# B&R Automation Studio project TD52 (part 134)

#### MsgSYCyclic.st
```iecst
(*******************************************************************************
MsgSY	 			 messages

This code is confidential and proprietary to the INNIO Company.
It may not be used in any form, or reproduced in any manner,
without written permission of the INNIO Company.
Copyright, INNIO Company, 2022

Customized modifications: -
------------------------

History:
-------
V2.12	24.04.2006	LH			adapted for esy new
V2.20	07.02.2007	LH			adapted for supporting customer mcb
		26.04.2007	LH			closing failure gcb (5th try was successful):
					               - gcb on + 10 sec --> reset counter
					               - dalay closing fail. = 11 sec
		09.05.2007	LH			0/1-sign. fail. mcbx: activation with RUN in case of old hardware
V2.30	18.01.2008	LH			adapted for test-bench run
		14.02.2008	LH			reset moved from end to begin
		28.03.2008	LH			gcb not closed and load > 10% --> gcb position failure
		07.04.2008	LH			new gcb position monitoring active with release from engine control
V2.311a	13.05.2008	LH			set delay time new gcb position failure up to 2 sec.
V2.33.0	16.07.2008	lettenb.	mcb[1].alm_psf disabled with PRF_I (circuitus)
V2.60.0	13.08.2009	lettenb.	ton_gcb_opf	for opening mcb with delay addedf
V3.20.0	14.04.2010	lettenb.	change to new global structure ALM
		11.11.2010				1216 enable busbar 1 voltage sensor failure	if not bSynch
		07.12.2010				1219 ctd_gcb_cf[1].LOAD	mit quitt_wa
								(reset ctd_gcb_cf[1] funktioniert nicht wenn eng[1].sy_rdy = false)
V3.99.0	25.02.2012	lettenb.	3329,3352,3575,3576,3577 added (integration V3.30-V3.40)
		24.05.2013				reset OUT_xx.txx2AB.bGnlTripx changed
		18.06.2013				2140 removed (made in MM_OP), 2139 logic changed, xMsg2139+xMsg2140 removed
V4.00.0	27.02.2014				logger added
		06.03.2014				Para.bGlowIgnPrevent -> Para.bGlowIgnPrevActive
		20.06.2014				VIS2MM.bServiceBegin --> IN_SY.bServiceMode (no 2nd plc-tag)
V4.00.1	19.11.2014				1042 generator power signal overload, without delay, new parameter(920 stapelfeld),
								1041 generator power signal missing (920 stapelfeld)
								1175,1216,1217,1220 enable with IN_SY.tPB2MM.bSys_Run
								1039 xTOF_SYANW removed, bugfix
V4.03.0	22.07.2015				2692,2693,2801 new, dyn.gridcode III(thaler)
                                2730 Temperature max generator switch gear
								init: xMsg1038 removed(see MM_GC)
		21.09.2015				2688 added + bugfix 1.5 -> 0.5
        04.02.2016				1041 xTON_LSA.PT for 920 from 0s -> 300ms to avoid 1041 at grid code event
V4.04.0	04.07.2016				2901-2903 added, tLockEng_ClosCond.Do added
		13.09.2016				1041 xGR_MAX_LSA_LD.Gw 1.5 -> 2.0 bar for 920(request: spyra klaus)
		28.09.2016				3400 added, holland/belgien standard, plattner joh.
		07.10.2016				2801 logic changed acc.kiel validation(thalerj)
		30.03.2017				1210 AND NOT IN_SY.tMns_MDF.Di -> AND IN_SY.tMns_MDF.Di, bugfix
		07.04.2017				gcb.alarm MM2VIS.bMsg1214 removed, bugfix
V4.05.0 31.05.2017  lettenb.    reservation for mcb2/mains2 messages removed(comment)
                                2934 added, grid code logic
		22.01.2018	lettenb.	1175,1189,1216,3329 bParaSetupOk added TO avoid message at plc startup
		24.01.2018				1214 mcb.remote, 5" delay added(to avoid mcb-off at plc startup),(glantschnig)
V4.05.1	09.03.2018	Perktold,	delayed A1042 trip (only HiHi part), 100ms normal, 500ms when LVRT Event is detected (for 5s)
V4.06.0 21.09.2018  Perktold,   A1042 implemented 110% overload step 3s delay excluded bBDC_Emergency_OFF
		11.10.2018				A1041 generator power signal missing --> 1s delay for NOT Type9 and GEN2
V4.07.0	31.10.2018	lettenb.	2330,9244,9245 added
		12.02.2019				9244 delay 0s->30s
		26.02.2019	Perktold	Update A1042, removed 120% overload case (ECR E18-00283)
		02.05.2019	lettenb.	1237,1238 removed(not used/->OP), clean up
V4.09.0	17.10.2019	lettenb.	9304 added, protection test mapping
		16.03.2020	lettenb.	2688 only active with synch.pulse(not with gcb closing to dead busbar), bugfix
V4.10.0	23.11.2020	lettenb.	9331,2354 added
		22.12.2020	lettenb.	1041: RiskClass setting corr.acc.TI 1100-0111
		22.02.2021	Arnold		1042: include 120% 500ms overload trip in island mode
V4.11.0	07.07.2021	lettenb.	init xMsg2692.Num: 2693->2692, bugfix
		29.09.2021	lettenb.	9304 delay 100->300ms for correct assistant value transfer, bugfix
V4.12.0	02.05.2022	Schmidt		W2688 (high sync current) threshold increased from 50% to 75% of nominal current
		15.06.2022	lettenb.	3269,3296,3297 added, dead bb synch
		10.03.2023	lettenb.	2366: detection of multiple short GCB OnOff events(BR6: puffmini causes engine stop/restart)
V4.13.0	17.08.2023	lettenb.	dead bb synch, bugfixes(BR21/wasserer,schwab,lettenb.)
		26.09.2023	Farre,		LCB operating message when open (B9083) or closed (B9084)
		07.11.2023	Hohensinner	added LV GCB op messages and warnings: B9085, W9382 and W9383
		29.11.2023	Goenczi,	W1175,W1189,W3412 reset, W1209 enable, W3412 set condition standardized
V4.14.0	25.10.2024	Farre,		GCB Opening Failure - W1217 and reverse power connected to GCB_OpF command (2024-241)

Instructions for use:
--------------------
1) declare alarm with function block "Alm"
	declare buffert alarm bit bMsg<message number>

2) use template to create a new alarm,
   substitue 0000 by alarm number and make settings:

	xMsg0000.Enable		:=	TRUE;		enable/disable alarm
	xMsg0000.Set		:=	FALSE;		alarm set condition
	xMsg0000.PT			:=	T#0s;		alarm delay time
	xMsg0000.Prio		:=	1;			alarm priority: 1-3 = trip, 4 = warning
	xMsg0000.RiskClass	:=	3;			risk class for remote alarm reset
	xMsg0000.Reset		:=	FALSE;		FALSE: for all standard alarms	prio 1,2,3 and warnings prio 4
										TRUE : for autoreset alarms

	bMsg0000			:=	xMsg0000.Q;	connect buffert alarm bit for VIS and control

3)  expand INIT

4)	include datapoint into OPC configuration for vis

(******************************************************************************
alarms overview:
W 1209 - 1215	mcb alarms
W 1216			general alarms sy
W 1217 - 1224	gcb alarms
*****************************************************************************

Outstandings:
------------
(*******************************************************************************)
PROGRAM _CYCLIC

	(* reset general trip *)
	OUT_SY.tSY2AB.bGnlTrip1		:=	FALSE;
	OUT_SY.tSY2AB.bGnlTrip2		:=	FALSE;
	OUT_SY.tSY2AB.bGnlTrip3		:=	FALSE;
	OUT_SY.tSY2AB.bGnlWarning	:=	FALSE;
	OUT_SY.tSY2AB.bTriptype1	:=	FALSE;
	OUT_SY.tSY2AB.bTriptype2	:=	FALSE;
	OUT_SY.tSY2AB.bTriptype3	:=	FALSE;

	(*---------------------------------------------------------------------------*)
	(* A1039 synchronizing failure *)
	xTON_SYST1(IN:=(OUT_SY.bSynchDem OR gcb.dmnd_sy OR mcb.dmnd_sy)
			AND 	IN_SY.tRel_Sync_Load.Do
			AND NOT IN_SY.tGCB_On.Di
			AND NOT bGnlTrip, PT:= T#600s);  // AT16

	xTON_SYST2(IN:= IN_SY.tEng_Run.Do AND NOT IN_SY.tGCB_On.Di, PT:= T#1200s); // AT32

	xMsg1039.Enable		:= TRUE;
	xMsg1039.Set		:= xTON_SYST1.Q OR xTON_SYST2.Q;
	xMsg1039.PT			:= T#0s;
	xMsg1039.Prio		:= 2;
	xMsg1039.RiskClass	:= 0;
	xMsg1039.Reset		:= FALSE;
	xMsg1039();
	MM2VIS.bMsg1039		:= xMsg1039.Q;

	(* A1041 generator power signal missing *)
 	(* generator power low *)
	xGR_MINR_P_Lo(In:= IN_SY.rP_Act_Norm, Gw:= Para.rP_LimLo, Hy:= Para.rP_HyLo);
	bP_Lo  := xGR_MINR_P_Lo.Q AND IN_SY.tPB2MM.bParaSetupOk;

	xTOF_bGen2_Act(IN := IN_SY.bGen2_Act, PT := T#5s);		//GEN2 Controller running + TOF delay for shutdown

	IF IN_SY.bMMD_GenAlarmTestOn THEN
		IF xEngType.Type9 THEN
			xTON_LSA(IN:= bP_Lo,                          										PT:= T#300ms);
		ELSIF NOT xEngType.Type9 AND xTOF_bGen2_Act.Q THEN
			xTON_LSA(IN:= bP_Lo,                                           						PT:= T#1s);
		ELSE
			xTON_LSA(IN:= bP_Lo,                                                               	PT:= T#15s);
		END_IF;
	ELSE
		IF xEngType.Type9 THEN
			xTON_LSA(IN:= bP_Lo AND NOT IN_SY.bEng_Dem_EPS AND bOMSS_Aut AND IN_SY.tGCB_On.Di, PT:= T#300ms);
		ELSIF NOT xEngType.Type9 AND xTOF_bGen2_Act.Q THEN
			xTON_LSA(IN:= bP_Lo AND NOT IN_SY.bEng_Dem_EPS AND bOMSS_Aut AND IN_SY.tGCB_On.Di, PT:= T#1s);
		ELSE
			xTON_LSA(IN:= bP_Lo AND NOT IN_SY.bEng_Dem_EPS AND bOMSS_Aut AND IN_SY.tGCB_On.Di, PT:= T#15s);
		END_IF;
	END_IF;

	(* Charge pressure higher than 1.5 bar / 2.0 bar(920) *)
	IF xEngType.Type9 THEN xGR_MAX_LSA_LD(In:= MAX(IN_SY.tPr_Ch_P2s.Ai, MAX(IN_SY.tPr_Ch_P2s_A.Ai, IN_SY.tPr_Ch_P2s_B.Ai)), Gw:= 2.0, Hy:= 0.01);
	ELSE                   xGR_MAX_LSA_LD(In:= MAX(IN_SY.tPr_Ch_P2s.Ai, MAX(IN_SY.tPr_Ch_P2s_A.Ai, IN_SY.tPr_Ch_P2s_B.Ai)), Gw:= 1.5, Hy:= 0.01);
	END_IF;
	xTON_LSA_LD(IN:= xGR_MAX_LSA_LD.Q, PT:= T#1s);

	xMsg1041.Enable		:= TRUE;
	IF IN_SY.bMMD_GenAlarmTestOn THEN	xMsg1041.Set :=	xTON_LSA.Q;
	ELSIF xEngType.Type9 OR xTOF_bGen2_Act.Q THEN	xMsg1041.Set :=	xTON_LSA.Q
											 		AND NOT bGnlTrip1
													AND NOT bGnlTrip2
								            		AND 	xTON_LSA_LD.Q
											 		AND(NOT IN_SY.bSCO_Active OR NOT Para.bGlowIgnPrevActive);
	ELSE									xMsg1041.Set :=	xTON_LSA.Q
								            		AND 	xTON_LSA_LD.Q
											 		AND(NOT IN_SY.bSCO_Active OR NOT Para.bGlowIgnPrevActive);
	END_IF;
	xMsg1041.PT			:= T#0s;
	xMsg1041.Prio		:= 2;
	xMsg1041.RiskClass	:= 3;
	xMsg1041.Reset		:= FALSE;
	xMsg1041();
	MM2VIS.bMsg1041 	:= xMsg1041.Q;
	bMsg1041_Test		:= xMsg1041.Test;
	MM2VIS.bMsg1041Set 	:= xMsg1041.Set;
	OUT_SY.bMsg1041Set  := xMsg1041.Set;

	(* A1042 generator power signal overload *)

	(*110% overload step 3s delay*)
	xGR_MAXR_P_Hi110  (In:= IN_SY.rP_Act_Norm_Filt, Gw:= 1.1,   Hy:= 0.01);
	xTON_P_Hi110(IN:= xGR_MAXR_P_Hi110.Q, PT:= T#3s);

	(*105% overload step 15s delay*)
	xGR_MAXR_P_Hi  (In:= IN_SY.rP_Act_Norm_Filt, Gw:= Para.rP_LimHi,   Hy:= Para.rP_HyHi);
	xTON_P_Hi(IN:= xGR_MAXR_P_Hi.Q, PT:= T#15s);

	(* 120% overload step 500ms delay - only in island mode*)
	xTON_ParaInit_P_LimHiHi(IN := IN_SY.tPB2MM.bParaSetupOk AND Para.rP_LimHiHi 		<= 0.0,	PT := T#1s500ms);
	xTON_ParaInit_Ti_P_LimHiHi(IN := IN_SY.tPB2MM.bParaSetupOk AND Para.ti_P_LimHiHi 	<= T#0s, PT := T#1s500ms);
	IF xTON_ParaInit_P_LimHiHi.Q THEN		Para.rP_LimHiHi 	:= 1.2;			END_IF;
	IF xTON_ParaInit_Ti_P_LimHiHi.Q THEN	Para.ti_P_LimHiHi 	:= T#500ms;		END_IF;

	xGR_MAXR_P_HiHi(In:= IN_SY.rP_Act_Norm,      Gw:= Para.rP_LimHiHi, Hy:= Para.rP_HyHi);
	xTON_P_HiHi(IN:= xGR_MAXR_P_HiHi.Q AND xOpMode.Island, PT:= Para.ti_P_LimHiHi);

	xMsg1042.Enable		:=	TRUE;
	xMsg1042.Set		:= IN_SY.tPB2MM.bParaSetupOk AND(xTON_P_Hi.Q OR xTON_P_Hi110.Q OR xTON_P_HiHi.Q);
	xMsg1042.PT			:=	T#0s;
	xMsg1042.Prio		:=	2;
	xMsg1042.RiskClass	:=	4;
	xMsg1042.Reset		:=	FALSE;
	xMsg1042();
	MM2VIS.bMsg1042		:=	xMsg1042.Q;
	bMsg1042_Test		:=	xMsg1042.Test;
	MM2VIS.bMsg1042Set	:=	xMsg1042.Set;
	OUT_SY.bMsg1042Set  :=  xMsg1042.Set;

	(* W1175 mains failure *)
	xMsg1175.Enable		:= IN_SY.tPB2MM.bParaSetupOk;
	xMsg1175.Set		:=(NOT OUT_SY.bMainsReturn OR NOT OUT_SY.bMnsOk) AND NOT OUT_SY.bRel_Island;
	xMsg1175.PT			:= T#0s;
	xMsg1175.Prio		:= 4;
	xMsg1175.RiskClass	:= 4;
	xMsg1175.Reset		:= IN_SY.bSetIslandMode;
	xMsg1175();
	MM2VIS.bMsg1175		:= xMsg1175.Q;

	(* W1189 release from synchronization missing *)
	xMsg1189.Enable		:= IN_SY.tPB2MM.bParaSetupOk;
	xMsg1189.Set		:= 		IN_SY.tPB2MM.bSys_Run
						AND NOT OUT_SY.bRelEngOpFromSy
						AND(	NOT OUT_SY.bOnly_Island
						  	OR		IN_SY.bEng_RPSDem
	                       	OR	NOT bN_EngStart1);
	xMsg1189.PT			:= T#0s;
	xMsg1189.Prio		:= 4;
	xMsg1189.RiskClass	:= 4;
	xMsg1189.Reset		:= IN_SY.bSetFixedPwrMode;
	xMsg1189();
	MM2VIS.bMsg1189		:= xMsg1189.Q;

	bN_EngStart1 := bN_EngStart;	(* delay of 1 cycle, to avoid alarm 1189 at normal shutdown with only island operation *)

	(* W1209 main circuit breaker position signal failure*)
	xMsg1209.Enable		:=  Para.bSyActive
					AND	   (Para.bMCB_Enable OR Para.bMCB_Ctr_Cust OR Para.bIslandOp_Enable OR Para.bOnlyIsland_Enable OR Para.bMSy)
					AND NOT OUT_SY.bTestBenchModeIsland
					AND NOT (Para.iSel_Customer = 2);
	xMsg1209.Set		:= IN_SY.tPB2MM.bSys_Run
					AND(   (    mcb.on AND     mcb.off)
						OR (NOT	mcb.on AND NOT mcb.off));
	xMsg1209.PT			:= T#5s;
	xMsg1209.Prio		:= 4;
	xMsg1209.RiskClass	:= 4;
	xMsg1209.Reset		:= FALSE;
	xMsg1209();
	MM2VIS.bMsg1209		:= xMsg1209.Q;

	(* W1210 main circuit breaker opening failure *)
	xMsg1210.Enable		:= Para.bSyActive AND Para.bMCB_Enable;
	xMsg1210.Set		:= mcb.on
					AND	NOT	MM2VIS.bMsg1210
					AND(	mcb.command_off
						OR (mcb.rel_trip AND IN_SY.tMns_MDF.Di AND NOT mains.ok));

	xMsg1210.PT			:= T#5s;
	xMsg1210.Prio		:= 4;
	xMsg1210.RiskClass	:= 4;
	xMsg1210.Reset		:= FALSE;
	xMsg1210();
	MM2VIS.bMsg1210		:= xMsg1210.Q;

	(* W1211 main circuit breaker switch closing failure *)
	r_trig_mcb_on(CLK:= mcb.command_on OR mcb.on);

	ton_mcb_on(IN:= mcb.on, PT:= T#60s);

	r_trig_mcb_ct(CLK:=	ton_mcb_on.Q
					OR	NOT	IN_SY.tPB2MM.bSys_Run
					OR	NOT	mcb.remote
					OR     (mcb.alm_cf	AND	IN_SY.tAB2SY.bResetWarning));

	ctd_mcb_cf.CD	:=	r_trig_mcb_on.Q	AND	mcb.remote;
	ctd_mcb_cf.LOAD	:=	r_trig_mcb_ct.Q;
	ctd_mcb_cf.PV	:=	5;
	ctd_mcb_cf();

	ton_ctd_mcb(IN := ctd_mcb_cf.Q, PT:= T#1s);
	ton_mcb_cf(IN:= mcb.rel_sy_puls AND NOT mcb.on, PT := T#600s);
	ton_mcb_cf1(IN:= mcb.command_on AND NOT mcb.on, PT := T#6s);

	xMsg1211.Enable		:= Para.bSyActive AND Para.bMCB_Enable;
	xMsg1211.Set		:= ton_ctd_mcb.Q	OR	ton_mcb_cf.Q	OR	ton_mcb_cf1.Q;
	xMsg1211.PT			:= T#0s;
	xMsg1211.Prio		:= 4;
	xMsg1211.RiskClass	:= 4;
	xMsg1211.Reset		:= FALSE;
	xMsg1211();
	MM2VIS.bMsg1211		:= xMsg1211.Q;

	(* W1212 mains circuit breaker 0-signal failure *)
	xMsg1212.Enable		:= Para.bSyActive AND Para.bMCB_Enable;
	xMsg1212.Set		:= 	IN_SY.tMCB_SM.Di
					AND		mcb.remote
					AND NOT mcb.rel_sy_puls
					AND NOT mcb.command_on;

	xMsg1212.PT			:= T#5s;
	xMsg1212.Prio		:= 4;
	xMsg1212.RiskClass	:= 4;
	xMsg1212.Reset		:= FALSE;
	xMsg1212();
	MM2VIS.bMsg1212		:= xMsg1212.Q;

	(* W1213 mains circuit breaker 1-signal failure *)
	xMsg1213.Enable		:= Para.bSyActive AND Para.bMCB_Enable;
	xMsg1213.Set		:=	NOT	IN_SY.tMCB_SM.Di
						AND		mcb.remote
						AND    (mcb.rel_sy_puls OR mcb.command_on);

	xMsg1213.PT			:= T#5s;
	xMsg1213.Prio		:= 4;
	xMsg1213.RiskClass	:= 4;
	xMsg1213.Reset		:= FALSE;
	xMsg1213();
	MM2VIS.bMsg1213		:= xMsg1213.Q;

	(* W1214 main circuit breaker overload/short-circuit *)
	xMsg1214.Enable		:= Para.bMCB_Enable OR Para.bMCB_Ctr_Cust;
	xMsg1214.Set		:=	NOT IN_SY.tMCB_OL.Di
				 		AND		mcb.remote;
	xMsg1214.PT			:= T#5s;
	xMsg1214.Prio		:= 4;
	xMsg1214.RiskClass	:= 4;
	xMsg1214.Reset		:= FALSE;
	xMsg1214();
	MM2VIS.bMsg1214		:= xMsg1214.Q;

	(* W1216 bus bar voltage sensor failure *)
	xMsg1216.Enable		:= IN_SY.tPB2MM.bParaSetupOk;
	xTOF1216(IN:= gcb.mdl OR IN_SY.tDemGenExcOff.Di, PT:= T#5s);
	IF Para.bSyActive THEN
		xMsg1216.Set	:= 	NOT	bb_alive
						AND(   (mcb.on				AND		mains.ok)
							OR (any_gcb_on_bb		AND	NOT	OUT_SY.bGen_Exc_Off AND NOT xTOF1216.Q));
	ELSE
		xMsg1216.Set	:=	NOT	IN_SY.tBB_Alive.Di
						AND(   (mcb.on				AND		mains.ok)
							OR (IN_SY.tGCB_On.Di	AND	NOT	OUT_SY.bGen_Exc_Off AND NOT xTOF1216.Q)
							OR  IN_SY.tC_CB_On.Di);
	END_IF;
	xMsg1216.PT			:= T#5s;
	xMsg1216.Prio		:= 4;
	xMsg1216.RiskClass	:= 4;
	xMsg1216.Reset		:= FALSE;
	xMsg1216();
	MM2VIS.bMsg1216		:= xMsg1216.Q;

	(* W1217 Generator circuit breaker position signal failure *)
	ton_gcb_psf(IN:=   (    gcb.on	AND		gcb.off)
					OR (NOT	gcb.on	AND	NOT gcb.off), PT:= T#3s);

	xMsg1217.Enable		:= Para.bSyActive AND IN_SY.tPB2MM.bSys_Run;
	xMsg1217.Set		:=  ton_gcb_psf.Q
					OR (NOT	gcb.on 	AND	NOT	bP_Lo AND IN_SY.tPB2MM.bParaSetupOk);
	xMsg1217.PT			:= T#2s;
	xMsg1217.Prio		:= 4;
	xMsg1217.RiskClass	:= 4;
	xMsg1217.Reset		:= FALSE;
	xMsg1217();
	MM2VIS.bMsg1217		:= xMsg1217.Q;

	OUT_SY.bGCB_psf_EngStop	:=	MM2VIS.bMsg1217 AND xOpMode.Stop;	(* send GCB position signal failure to Opstate - Block module release sync missing *)

	(* W1218 generator circuit breaker opening failure *)
	xTON_gcb_psf_P_rev	(IN:= IN_SY.bPact_Rev AND xMsg1217.Q, PT:= T#5s);	(* Pact negative and gcb position failure detected *)

	xMsg1218.Enable		:= Para.bSyActive;
	xMsg1218.Set		:=  (gcb.on AND (gcb.command_off	OR	NOT	IN_SY.tRel_Sync_Load.Do))
						OR	xTON_gcb_psf_P_rev.Q;			(* include in opening failure when reverse power is measured *)

	xMsg1218.PT			:= T#5s;
	xMsg1218.Prio		:= 4;
	xMsg1218.RiskClass	:= 4;
	xMsg1218.Reset		:= FALSE;
	xMsg1218();
	MM2VIS.bMsg1218		:= xMsg1218.Q;

	gcb.alm_opf			:= xMsg1218.Q;

	ton_gcb_opf.IN 		:= 	(gcb.alm_opf AND NOT gcb.off) 	(* GCB opening failure - gcb_on and command_off but gcb_off response is false *)
						OR 	xTON_gcb_psf_P_rev.Q;			(* GCB position failure - gcb_on and gcb_off or not gcb_on and not gcb_off, when reverse power *)
	ton_gcb_opf.PT 		:= 	T#2s;
	ton_gcb_opf();
	gcb_opf_delay		:=	ton_gcb_opf.Q;	(* opening mcb after delay *)

	(* W1219 generator circuit breaker closing failure *)
	r_trig_gcb_on(CLK:= IN_SY.tGCB_SM1.Di);
	ton_gcb_on(IN:=	gcb.on, PT:= T#10s);
	r_trig_gcb_ct(CLK:= NOT IN_SY.tRel_Sync_Load.Do OR ton_gcb_on.Q);

	ctd_gcb_cf.CD	:=	r_trig_gcb_on.Q;
	ctd_gcb_cf.LOAD	:=	r_trig_gcb_ct.Q OR IN_SY.tAB2SY.bResetWarning;
	ctd_gcb_cf.PV	:=	5;
	ctd_gcb_cf();

	ton_ctd_gcb(IN:=	ctd_gcb_cf.Q, PT:= T#11s);
	ton_gcb_cf1(IN:=	gcb.command_on AND NOT gcb.on, PT:= T#5s);

	xMsg1219.Enable		:= Para.bSyActive;
	xMsg1219.Set		:= (ton_ctd_gcb.Q OR ton_gcb_cf1.Q) AND NOT MM2VIS.bMsg2366;
	xMsg1219.PT			:= T#0s;
	xMsg1219.Prio		:= 4;
	xMsg1219.RiskClass	:= 4;
	xMsg1219.Reset		:= FALSE;
	xMsg1219();
	MM2VIS.bMsg1219		:= xMsg1219.Q;

	(* W1220 generator circuit breaker 0-signal failure *)
	xMsg1220.Enable		:= Para.bSyActive AND IN_SY.tPB2MM.bSys_Run;
	xMsg1220.Set		:= (	IN_SY.tGCB_SM1.Di	    AND NOT	gcb.release)												(* SM1 *)
						OR (NOT	IN_SY.tRel_Sync_Load.Do AND	NOT	gcb.dmnd_sy AND	NOT	gcb.release AND	NOT	IN_SY.tGCB_SM2.Di);	(* SM2 *)
	xMsg1220.PT			:= T#5s;
	xMsg1220.Prio		:= 4;
	xMsg1220.RiskClass	:= 4;
	xMsg1220.Reset		:= FALSE;
	xMsg1220();
	MM2VIS.bMsg1220		:= xMsg1220.Q;

	(* W1221 generator circuit breaker 1-signal failure *)
	xMsg1221.Enable		:= Para.bSyActive;
	xMsg1221.Set		:= (gcb.on AND NOT gcb.command_off AND NOT IN_SY.tGCB_SM1.Di)
						OR (IN_SY.tRel_Sync_Load.Do	AND	IN_SY.tGCB_SM2.Di);
	xMsg1221.PT			:= T#5s;
	xMsg1221.Prio		:= 4;
	xMsg1221.RiskClass	:= 4;
	xMsg1221.Reset		:= FALSE;
	xMsg1221();
	MM2VIS.bMsg1221		:= xMsg1221.Q;

	(* W1222 generator manual circuit breaker opened *)
	xMsg1222.Enable		:= FALSE;
	xMsg1222.Set		:= NOT gcb.rdy;
	xMsg1222.PT			:= T#0s;
	xMsg1222.Prio		:= 4;
	xMsg1222.RiskClass	:= 4;
	xMsg1222.Reset		:= FALSE;
	xMsg1222();
	MM2VIS.bMsg1222		:= xMsg1222.Q;

    (* A2330 mid voltage CB failure *)
	xMsg2330.Enable		:= TRUE;
	xMsg2330.Set		:= NOT IN_SY.tMidVoltCB_Failure.Di;
	xMsg2330.PT			:= T#0s;
	xMsg2330.Prio		:= 2;
	xMsg2330.RiskClass	:= 4;
	xMsg2330.Reset		:= FALSE;
	xMsg2330();
	MM2VIS.bMsg2330		:= xMsg2330.Q;

	(* A2354 Earth fault bus bar *)
	xMsg2354.Enable    := TRUE;
	xMsg2354.Set       := NOT IN_SY.tGndFault_BB.Di;
	xMsg2354.PT        := T#0s;
	xMsg2354.RiskClass := 4;
	xMsg2354.Prio      := 2;
	xMsg2354.Reset     := FALSE;
	xMsg2354();
	MM2VIS.bMsg2354    := xMsg2354.Q;

	(* A2366 Generator circuit breaker closing failure *)
	(* detection of multiple short GCB OnOff events (BR6: puffmini causes engine stop/restart) *)
	xTP_gcb_on (IN:=     IN_SY.tGCB_On.Di, PT:= T#1s);
	xF_TRIG_gcb_on(CLK:= IN_SY.tGCB_On.Di);
	xR_TRIG_gcb_OnOffct(CLK:= ton_gcb_on.Q);

	xCTD_gcb_OnOffEvent.CD   :=	xTP_gcb_on.Q AND xF_TRIG_gcb_on.Q;
	xCTD_gcb_OnOffEvent.LOAD :=	xR_TRIG_gcb_OnOffct.Q OR MM2VIS.bMsg2366 OR EDGEPOS(IN_SY.tPB2MM.bParaSetupOk);
	xCTD_gcb_OnOffEvent.PV   :=	5;
	xCTD_gcb_OnOffEvent();

	xMsg2366.Enable    := IN_SY.tPB2MM.bParaSetupOk;
	xMsg2366.Set       := xCTD_gcb_OnOffEvent.Q;
	xMsg2366.PT        := T#0s;
	xMsg2366.RiskClass := 4;
	xMsg2366.Prio      := 3;
	xMsg2366.Reset     := FALSE;
	xMsg2366();
	MM2VIS.bMsg2366    := xMsg2366.Q;

	(* W2688 Generator current at synchronization too high *)
	xTP_GCB_On(IN:= IN_SY.tGCB_On.Di, PT:= T#10s);
	xTP_MMD_SynchDO(IN:= IN_SY.bMMD_SynchDO[1], PT:= T#10s);

	xMsg2688.Enable    := TRUE;
	xMsg2688.Set       := xTP_GCB_On.Q
					AND   xTP_MMD_SynchDO.Q
				    AND ((IN_SY.rI_MaxL1[1] > (0.75 * Para.rI_GenNom[1]))
					  OR (IN_SY.rI_MaxL2[1] > (0.75 * Para.rI_GenNom[1]))
					  OR (IN_SY.rI_MaxL3[1] > (0.75 * Para.rI_GenNom[1])));
	xMsg2688.PT        := T#0s;
	xMsg2688.RiskClass := 4;
	xMsg2688.Prio      := 4;
	xMsg2688.Reset     := FALSE;
	xMsg2688();
	MM2VIS.bMsg2688    :=  xMsg2688.Q;

	(* W2692 mains circuit breaker opening failure *)
	xMsg2692.Enable		:= TRUE;
	xMsg2692.Set		:= NOT IN_SY.tMCB_OpF_Ext.Di;
	xMsg2692.PT			:= T#0s;
	xMsg2692.Prio		:= 4;
	xMsg2692.RiskClass	:= 4;
	xMsg2692.Reset		:= FALSE;
	xMsg2692();
	MM2VIS.bMsg2692		:= xMsg2692.Q;

	(* W2693 generator circuit breaker opening failure *)
	xMsg2693.Enable		:= TRUE;
	xMsg2693.Set		:= NOT IN_SY.tGCB_OpF_Ext.Di;
	xMsg2693.PT			:= T#0s;
	xMsg2693.Prio		:= 4;
	xMsg2693.RiskClass	:= 4;
	xMsg2693.Reset		:= FALSE;
	xMsg2693();
	MM2VIS.bMsg2693		:= xMsg2693.Q;

        (* W2730 low voltage CB failure *)	(* high temperature NLD / BEL specific *)
	xMsg2730.Enable		:= Para.bP_Red_TempMax_GenCB_Active;
	xMsg2730.Set		:= NOT IN_SY.tTempMax_GenCB.Di;
	xMsg2730.PT			:= T#0s;
	xMsg2730.Prio		:= 4;
	xMsg2730.RiskClass	:= 4;
	xMsg2730.Reset		:= FALSE;
	xMsg2730();
	MM2VIS.bMsg2730		:= xMsg2730.Q;

	(* W3329 earth circuit breaker closed *)	(* france country specific *)
	xMsg3329.Enable		:= IN_SY.tPB2MM.bParaSetupOk;
	xMsg3329.Set		:= NOT IN_SY.tEarthCB_Off.Di;
	xMsg3329.PT			:= T#0s;
	xMsg3329.Prio		:= 2;
	xMsg3329.RiskClass	:= 4;
	xMsg3329.Reset		:= FALSE;
	xMsg3329();
	MM2VIS.bMsg3329		:= xMsg3329.Q;

	(* W3352 earth circuit breaker opened *)	(* france country specific *)
	xMsg3352.Enable		:= TRUE;
	xMsg3352.Set		:= NOT IN_SY.tIsoCB_Off.Di;
	xMsg3352.PT			:= T#0s;
	xMsg3352.Prio		:= 2;
	xMsg3352.RiskClass	:= 4;
	xMsg3352.Reset		:= FALSE;
	xMsg3352();
	MM2VIS.bMsg3352		:= xMsg3352.Q;

	(* A3400 module blocked by no operating release from sy or cooling water temp.low *)
	xMsg3400.Enable		:= (Para.iCountry = iHolland);
	xMsg3400.Set		:=  NOT OUT_SY.bRelEngOpFromSy
						OR( 	bOMSS_Aut AND IN_SY.bT_ECW_Lo);
	xMsg3400.PT			:= T#0s;
	xMsg3400.Prio		:= 0;	 (* special for holland/plattner joh. *)
	xMsg3400.RiskClass	:= 4;
	xMsg3400.Reset		:= TRUE; (* auto reset *)
	xMsg3400();
	MM2VIS.bMsg3400		:= xMsg3400.Q;

	(* W3412 mains monitoring device failure/ generator protection relay failure *)
	xMsg3412.Enable		:= TRUE;
	xMsg3412.Set		:= NOT IN_SY.tMns_MDF.Di AND NOT IN_SY.bSetIslandMode;
	xMsg3412.PT			:= T#0s;
	xMsg3412.Prio		:= 4;
	xMsg3412.RiskClass	:= 4;
	xMsg3412.Reset		:= IN_SY.bSetIslandMode;
	xMsg3412();
	MM2VIS.bMsg3412		:= xMsg3412.Q;

	(* W3575 mains failure GTE2666 *)	(* france country specific *)
	xMsg3575.Enable		:= TRUE;
	xMsg3575.Set		:= NOT IN_SY.tMnsOk_GTE.Di;
	xMsg3575.PT			:= T#0s;
	xMsg3575.Prio		:= 4;
	xMsg3575.RiskClass	:= 4;
	xMsg3575.Reset		:= FALSE;
	xMsg3575();
	MM2VIS.bMsg3575		:= xMsg3575.Q;

	(* W3576 mains failure C13.100 *)	(* france country specific *)
	xMsg3576.Enable		:= TRUE;
	xMsg3576.Set		:= NOT IN_SY.tMnsOk_TGS.Di;
	xMsg3576.PT			:= T#0s;
	xMsg3576.Prio		:= 4;
	xMsg3576.RiskClass	:= 4;
	xMsg3576.Reset		:= FALSE;
	xMsg3576();
	MM2VIS.bMsg3576		:= xMsg3576.Q;

	(* W3577 earth circuit breaker opened *)	(* france country specific *)
	xMsg3577.Enable		:= TRUE;
	xMsg3577.Set		:= NOT IN_SY.tMnsOk_C13100.Di;
	xMsg3577.PT			:= T#0s;
	xMsg3577.Prio		:= 4;
	xMsg3577.RiskClass	:= 4;
	xMsg3577.Reset		:= FALSE;
	xMsg3577();
	MM2VIS.bMsg3577		:= xMsg3577.Q;

	(* W9244 generator circuit breaker not ready *)
	xMsg9244.Enable		:= TRUE;
	xMsg9244.Set		:= NOT IN_SY.tGCB_Rdy.Di;
	xMsg9244.PT			:= T#30s;
	xMsg9244.Prio		:= 4;
	xMsg9244.RiskClass	:= 4;
	xMsg9244.Reset		:= FALSE;
	xMsg9244();
	MM2VIS.bMsg9244		:= xMsg9244.Q;

	(* W9245 generator circuit breaker not racked-in *)
	xMsg9245.Enable		:= TRUE;
	xMsg9245.Set		:= NOT IN_SY.tGCB_Rac.Di;
	xMsg9245.PT			:= T#0s;
	xMsg9245.Prio		:= 4;
	xMsg9245.RiskClass	:= 4;
	xMsg9245.Reset		:= FALSE;
	xMsg9245();
	MM2VIS.bMsg9245		:= xMsg9245.Q;

	(* W9304 generator circuit breaker closing time deviation high *)
	xMsg9304.Enable		:= Para.bMMDSynch_Act[1] AND IN_SY.tPB2MM.bParaSetupOk;
	xMsg9304.Set		:= bGCBctd;
	xMsg9304.PT			:= T#300ms;(* delay needed for assistant value transfer(tiGCB_ClosTimeOld) to HMI *)
	xMsg9304.Prio		:= 4;
	xMsg9304.RiskClass	:= 4;
	xMsg9304.Reset		:= TRUE;(* autoreset, because reset is done in task: gcbTC1 *)
	xMsg9304();
	MM2VIS.bMsg9304		:= xMsg9304.Q;

	(* W9331 maintenance request generator circuit breaker *)
	xMsg9331.Enable		:= IN_SY.tPB2MM.bParaSetupOk AND (Para.rU_Gen_Nom[1] < 1000);
	xMsg9331.Set		:= (VIS2MM.iGCB_OnCnt >= Para.iGCB_OnCnt_LimHi);
	xMsg9331.PT			:= T#0s;
	xMsg9331.Prio		:= 4;
	xMsg9331.RiskClass	:= 4;
	xMsg9331.Reset		:= FALSE;
	xMsg9331();
	MM2VIS.bMsg9331		:= xMsg9331.Q;

	(* W9382 GCB contact wear over 80% *)
	xMsg9382.Enable		:= IN_SY.tPB2MM.bSys_Run;
	xMsg9382.Set		:= bW9382_GCB_Wear80;
	xMsg9382.PT			:= T#0s;
	xMsg9382.Prio		:= 4;
	xMsg9382.RiskClass	:= 4;
	xMsg9382.Reset		:= FALSE;
	xMsg9382();
	MM2VIS.bMsg9382		:= xMsg9382.Q;

	(* W9383 GCB contact wear over 95% *)
	xMsg9383.Enable		:= IN_SY.tPB2MM.bSys_Run;
	xMsg9383.Set		:= bW9383_GCB_Wear95;
	xMsg9383.PT			:= T#0s;
	xMsg9383.Prio		:= 4;
	xMsg9383.RiskClass	:= 4;
	xMsg9383.Reset		:= FALSE;
	xMsg9383();
	MM2VIS.bMsg9383		:= xMsg9383.Q;

	(*---------------------------------------------------------------------------*)
	(* mains circuit breaker alarms *)
	mcb.alm_psf		:=		MM2VIS.bMsg1209;
	mcb.alm_opf		:=		MM2VIS.bMsg1210;
	mcb.alm_cf		:=		MM2VIS.bMsg1211;
	mcb.alm_0sf 	:=		MM2VIS.bMsg1212;
	mcb.alm_1sf 	:=		MM2VIS.bMsg1213;
	mcb.alm_ol		:=		MM2VIS.bMsg1214;

	mcb.alarm		:=		MM2VIS.bMsg1209
						OR	MM2VIS.bMsg1210
						OR	MM2VIS.bMsg1211
						OR	MM2VIS.bMsg1212
						OR	MM2VIS.bMsg1213
						OR	MM2VIS.bMsg1214;

	(* generator circuit breaker alarms *)
	gcb.alm_psf		:=		MM2VIS.bMsg1217;
	gcb.alm_opf		:=		MM2VIS.bMsg1218;
	gcb.alm_cf		:=		MM2VIS.bMsg1219;
	gcb.alm_0sf 	:=		MM2VIS.bMsg1220;
	gcb.alm_1sf 	:=		MM2VIS.bMsg1221;
	gcb.alm_ol;

	gcb.alarm		:=		MM2VIS.bMsg1217
						OR	MM2VIS.bMsg1218
						OR	MM2VIS.bMsg1219
						OR	MM2VIS.bMsg1220
						OR	MM2VIS.bMsg1221
						OR	MM2VIS.bMsg1222;

	(*---------------------------------------------------------------------------*)
	(* operating messages > AMM *)

	(* B1235 generator circuit breaker closed *)
	xMsg1235.Enable		:=	TRUE;
	xMsg1235.Set		:=		IN_SY.tGCB_On.Di;
	xMsg1235.Reset		:=	TRUE;
	xMsg1235();
	MM2VIS.bMsg1235		:= xMsg1235.Q;

	(* B1236 generator circuit breaker opened *)
	xMsg1236.Enable		:=	IN_SY.tPB2MM.bSys_Run;
	xMsg1236.Set		:=	NOT IN_SY.tGCB_On.Di;
	xMsg1236.Reset		:=	TRUE;
	xMsg1236();
	MM2VIS.bMsg1236		:= xMsg1236.Q;

	(* B2139 synchronizing running  *)
	xMsg2139.Enable		:=	TRUE;
	xMsg2139.Set		:=	OUT_SY.bGCB_DemSy  AND NOT OUT_SY.bBB_dead;
	xMsg2139.Reset		:=	TRUE;
	xMsg2139();
	MM2VIS.bMsg2139		:= xMsg2139.Q;

	(* B2801 Module blocked by grid connection conditions *)
	xMsg2801.Enable		:=	TRUE;
//	xMsg2801.Set		:=  NOT bBBClosCond_Fault
//						AND	NOT bAMM_ClosCond_Ok
//						AND   ((IN_SY.bEng_Bloc AND NOT bN_EngStart)(* = iIdx_Eng_State = 19 = blocking module *)
//							OR  IN_SY.bMMD_BB_AlarmTestOn);

	xMsg2801.Set		:= (NOT bAMM_ClosCond_Ok AND NOT bBBClosCond_Fault AND(IN_SY.bEng_Bloc AND NOT bN_EngStart))(* = iIdx_Eng_State = 19 = blocking module *)
						OR (NOT bAMM_ClosCond_Ok AND     IN_SY.bMMD_BB_AlarmTestOn);

	xMsg2801.Reset		:=	TRUE;
	xMsg2801();
	MM2VIS.bMsg2801		:= xMsg2801.Q;
	OUT_SY.tLockEng_ClosCond.Do	:= NOT MM2VIS.bMsg2801;	//acc.kiel validation
	MM2VIS.bMsg2801Set	:= xMsg2801.Set;
	OUT_SY.bMsg2801Set  := xMsg2801.Set;

	(* B2901 synchronization selection OFF *)
	xMsg2901.Enable		:=	IN_SY.tPB2MM.bSys_Run;
	xMsg2901.Set		:=	bSyOMSS_Off;
	xMsg2901.Reset		:=	TRUE;
	xMsg2901();
	MM2VIS.bMsg2901		:= xMsg2901.Q;

	(* B2902 synchronization selection MAN *)
	xMsg2902.Enable		:=	IN_SY.tPB2MM.bSys_Run;
	xMsg2902.Set		:=	bSyOMSS_Man;
	xMsg2902.Reset		:=	TRUE;
	xMsg2902();
	MM2VIS.bMsg2902		:= xMsg2902.Q;

	(* B2903 synchronization selection AUT *)
	xMsg2903.Enable		:=	IN_SY.tPB2MM.bSys_Run;
	xMsg2903.Set		:=	bSyOMSS_Aut;
	xMsg2903.Reset		:=	TRUE;
	xMsg2903();
	MM2VIS.bMsg2903		:= xMsg2903.Q;

	(* B2934 Module blocked by grid connection conditions - after mains failure *)
	xMsg2934.Enable		:=	TRUE;
//	xMsg2934.Set		:=  bBBClosCond_Fault
//					AND NOT bAMM_ClosCond_Ok
//					AND   ((IN_SY.bEng_Bloc AND NOT bN_EngStart)(* = iIdx_Eng_State = 19 = blocking module *)
//	OR  IN_SY.bMMD_BB_AlarmTestOn);

	xMsg2934.Set		:= (NOT bAMM_AfMnsF_ClosCond_Ok AND bBBClosCond_Fault AND(IN_SY.bEng_Bloc AND NOT bN_EngStart))(* = iIdx_Eng_State = 19 = blocking module *)
						OR (NOT bAMM_AfMnsF_ClosCond_Ok AND IN_SY.bMMD_BB_AlarmTestOn);

	xMsg2934.Reset		:=	TRUE;
	xMsg2934();
	MM2VIS.bMsg2934		:= xMsg2934.Q;
	OUT_SY.tAfMnsF_LockEng_ClosCond.Do := NOT MM2VIS.bMsg2934;
	MM2VIS.bMsg2934Set	:= xMsg2934.Set;
	OUT_SY.bMsg2934Set	:= xMsg2934.Set;

	(* B3253 begin of maintenance/testbench mode *)
	xMsg3253.Enable		:=	TRUE;
	xMsg3253.Set		:=	bTestBenchMode OR IN_SY.bServiceMode;
	xMsg3253.Reset		:=	TRUE;
	xMsg3253();
	MM2VIS.bMsg3253		:=	xMsg3253.Q;

	(* B3254 end of maintenance/testbench mode *)
	xMsg3254.Enable		:=	IN_SY.tPB2MM.bSys_Run;
	xMsg3254.Set		:=	NOT bTestBenchMode AND NOT IN_SY.bServiceMode;
	xMsg3254.Reset		:=	TRUE;
	xMsg3254();
	MM2VIS.bMsg3254		:=	xMsg3254.Q;

	(* B3263 mains circuit breaker closed *)
	xMsg3263.Enable		:=	TRUE;
	xMsg3263.Set		:=		OUT_SY.bMCB_On;
	xMsg3263.Reset		:=	TRUE;
	xMsg3263();
	MM2VIS.bMsg3263		:=	xMsg3263.Q;

	(* B3264 mains circuit breaker opened *)
	xMsg3264.Enable		:=	IN_SY.tPB2MM.bSys_Run;
	xMsg3264.Set		:=	NOT OUT_SY.bMCB_On;
	xMsg3264.Reset		:=	TRUE;
	xMsg3264();
	MM2VIS.bMsg3264		:=	xMsg3264.Q;

	(* B3265 demand close GCB *)
	xMsg3265.Enable		:=	TRUE;
	xMsg3265.Set		:=	ton_gcb_dmnd_sy.IN AND OUT_SY.bBB_dead;
	xMsg3265.Reset		:=	TRUE;
	xMsg3265();
	MM2VIS.bMsg3265		:=	xMsg3265.Q;

	(* B3266 mains failure on *)
	xMsg3266.Enable		:=	IN_SY.tPB2MM.bSys_Run;
	xMsg3266.Set		:=	NOT OUT_SY.bMnsOk;
	xMsg3266.Reset		:=	TRUE;
	xMsg3266();
	MM2VIS.bMsg3266		:=	xMsg3266.Q;

	(* B3267 mains failure off *)
	xMsg3267.Enable		:=	IN_SY.tPB2MM.bSys_Run;
	xMsg3267.Set		:=		OUT_SY.bMnsOk;
	xMsg3267.Reset		:=	TRUE;
	xMsg3267();
	MM2VIS.bMsg3267		:=	xMsg3267.Q;

	(* B3269 generator de-energized *)
	xMsg3269.Enable		:=	IN_SY.tPB2MM.bSys_Run;
	xMsg3269.Set		:=	bGen_DeExc_Rdy;
	xMsg3269.Reset		:=	TRUE;
	xMsg3269();
	MM2VIS.bMsg3269		:=	xMsg3269.Q;

	(* B3296 demand generator excitation off *)
	xMsg3296.Enable		:=	IN_SY.tPB2MM.bSys_Run;
	xMsg3296.Set		:=	bGenDeexitDem;
	xMsg3296.Reset		:=	TRUE;
	xMsg3296();
	MM2VIS.bMsg3296		:=	xMsg3296.Q;

	(* B3297 demand generator excitation on *)
	xMsg3297.Enable		:=	IN_SY.tPB2MM.bSys_Run;
	xMsg3297.Set		:=	NOT bGenDeexitDem;
	xMsg3297.Reset		:=	TRUE;
	xMsg3297();
	MM2VIS.bMsg3297		:=	xMsg3297.Q;

	(* B9083 Line circuit breaker opened *)
	xMsg9083.Enable		:=	IN_SY.tLineCB_On.GoodQual;
	xMsg9083.Set		:=	NOT IN_SY.tLineCB_On.Di;
	xMsg9083.Reset		:=	TRUE;
	xMsg9083();
	MM2VIS.bMsg9083		:=	xMsg9083.Q;

	(* B9084 Line circuit breaker closed *)
	xTP_B9084(IN:= IN_SY.tLineCB_On.Di, PT:= T#20s);

	xMsg9084.Enable		:=	IN_SY.tLineCB_On.GoodQual;
	xMsg9084.Set		:=	xTP_B9084.Q;
	xMsg9084.Reset		:=	TRUE;
	xMsg9084();
	MM2VIS.bMsg9084		:=	xMsg9084.Q;

	(* B9085 Parameters saved to the GCB *)
	xMsg9085.Enable		:=	IN_SY.tPB2MM.bSys_Run;
	xMsg9085.Set		:=	bB9085_GCB_ParaSaved;
	xMsg9085.Reset		:=	TRUE;
	xMsg9085();
	MM2VIS.bMsg9085		:=	xMsg9085.Q;

(* B template
	xMsg.Enable		:=	TRUE;
	xMsg.Set		:=	bBool;
	xMsg.Reset		:=	TRUE;
	xMsg();
	MM2VIS.bMsg		:=	xMsg.Q;
	*)

	(*---------------------------------------------------------------------------*)
	(* general alarms for further module operations *)
	bGnlTrip1		:=	OUT_SY.tSY2AB.bGnlTrip1   OR IN_SY.tAB2SY.bGnlTrip1;
	bGnlTrip2		:=	OUT_SY.tSY2AB.bGnlTrip2   OR IN_SY.tAB2SY.bGnlTrip2;
	bGnlTrip3		:=	OUT_SY.tSY2AB.bGnlTrip3   OR IN_SY.tAB2SY.bGnlTrip3;
	bGnlWarning		:=	OUT_SY.tSY2AB.bGnlWarning OR IN_SY.tAB2SY.bGnlWarning;

	bGnlTrip		:=	bGnlTrip1 OR bGnlTrip2 OR bGnlTrip3;

(*******************************************************************************)
END_PROGRAM
```

#### MsgSYInit.st
```iecst
(*******************************************************************************
Msg_VE	 			 alarms generation MM_ventilation

This code is confidential and proprietary to the INNIO Company.
It may not be used in any form, or reproduced in any manner,
without written permission of the INNIO Company.
Copyright, INNIO Company, 2019

Customized modifications: -
------------------------

History:
-------
V0.00.0	29.07.2011	lettenb.	new

Instructions for use:
--------------------
1) declare alarm with function block "Msg"

2) use template to create a new alarm, substitue 0000 by message number:

	xMsg0000.Num		:=	0000;					alarm number
	xMsg0000.AmmSysAdr	:=  iAdrAmmBase2MM;			do not change
	xMsg0000.AmmOutAdr	:=  iAdrMM2AmmBase;			do not change

3) 	set alarm number

Outstandings:
------------
(*******************************************************************************)
PROGRAM _INIT

	iAdrAmmBase2MM		:=  ADR(IN_SY.tAB2SY);
	iAdrMM2AmmBase		:=  ADR(OUT_SY.tSY2AB);

	(*---------------------------------------------------------------------------*)
	xMsg1039.Num		:=  1039;
	xMsg1039.AmmInAdr	:=  iAdrAmmBase2MM;
	xMsg1039.AmmOutAdr	:=  iAdrMM2AmmBase;

	xMsg1041.Num		:=  1041;
	xMsg1041.AmmInAdr	:=  iAdrAmmBase2MM;
	xMsg1041.AmmOutAdr	:=  iAdrMM2AmmBase;

	xMsg1042.Num		:=  1042;
	xMsg1042.AmmInAdr	:=  iAdrAmmBase2MM;
	xMsg1042.AmmOutAdr	:=  iAdrMM2AmmBase;

	xMsg1109.Num		:=  1109;
	xMsg1109.AmmInAdr	:=  iAdrAmmBase2MM;
	xMsg1109.AmmOutAdr	:=  iAdrMM2AmmBase;

	xMsg1175.Num		:=  1175;
	xMsg1175.AmmInAdr	:=  iAdrAmmBase2MM;
	xMsg1175.AmmOutAdr	:=  iAdrMM2AmmBase;

	xMsg1189.Num		:=  1189;
	xMsg1189.AmmInAdr	:=  iAdrAmmBase2MM;
	xMsg1189.AmmOutAdr	:=  iAdrMM2AmmBase;

	xMsg1209.Num		:=  1209;
	xMsg1209.AmmInAdr	:=  iAdrAmmBase2MM;
	xMsg1209.AmmOutAdr	:=  iAdrMM2AmmBase;

	xMsg1210.Num		:=  1210;
	xMsg1210.AmmInAdr	:=  iAdrAmmBase2MM;
	xMsg1210.AmmOutAdr	:=  iAdrMM2AmmBase;

	xMsg1211.Num		:=  1211;
	xMsg1211.AmmInAdr	:=  iAdrAmmBase2MM;
	xMsg1211.AmmOutAdr	:=  iAdrMM2AmmBase;

	xMsg1212.Num		:=  1212;
	xMsg1212.AmmInAdr	:=  iAdrAmmBase2MM;
	xMsg1212.AmmOutAdr	:=  iAdrMM2AmmBase;

	xMsg1213.Num		:=  1213;
	xMsg1213.AmmInAdr	:=  iAdrAmmBase2MM;
	xMsg1213.AmmOutAdr	:=  iAdrMM2AmmBase;

	xMsg1214.Num		:=  1214;
	xMsg1214.AmmInAdr	:=  iAdrAmmBase2MM;
	xMsg1214.AmmOutAdr	:=  iAdrMM2AmmBase;

	xMsg1216.Num		:=  1216;
	xMsg1216.AmmInAdr	:=  iAdrAmmBase2MM;
	xMsg1216.AmmOutAdr	:=  iAdrMM2AmmBase;

	xMsg1217.Num		:=  1217;
	xMsg1217.AmmInAdr	:=  iAdrAmmBase2MM;
	xMsg1217.AmmOutAdr	:=  iAdrMM2AmmBase;

	xMsg1218.Num		:=  1218;
	xMsg1218.AmmInAdr	:=  iAdrAmmBase2MM;
	xMsg1218.AmmOutAdr	:=  iAdrMM2AmmBase;

	xMsg1219.Num		:=  1219;
	xMsg1219.AmmInAdr	:=  iAdrAmmBase2MM;
	xMsg1219.AmmOutAdr	:=  iAdrMM2AmmBase;

	xMsg1220.Num		:=  1220;
	xMsg1220.AmmInAdr	:=  iAdrAmmBase2MM;
	xMsg1220.AmmOutAdr	:=  iAdrMM2AmmBase;

	xMsg1221.Num		:=  1221;
	xMsg1221.AmmInAdr	:=  iAdrAmmBase2MM;
	xMsg1221.AmmOutAdr	:=  iAdrMM2AmmBase;

	xMsg1222.Num		:=  1222;
	xMsg1222.AmmInAdr	:=  iAdrAmmBase2MM;
	xMsg1222.AmmOutAdr	:=  iAdrMM2AmmBase;

	xMsg1235.Num		:=	1235;
	xMsg1235.AmmInAdr	:=  iAdrAmmBase2MM;
	xMsg1235.AmmOutAdr	:=  iAdrMM2AmmBase;

	xMsg1236.Num		:=	1236;
	xMsg1236.AmmInAdr	:=  iAdrAmmBase2MM;
	xMsg1236.AmmOutAdr	:=  iAdrMM2AmmBase;

	xMsg2139.Num		:=	2139;
	xMsg2139.AmmInAdr	:=  iAdrAmmBase2MM;
	xMsg2139.AmmOutAdr	:=  iAdrMM2AmmBase;

	xMsg2330.Num		:=	2330;
	xMsg2330.AmmInAdr	:=  iAdrAmmBase2MM;
	xMsg2330.AmmOutAdr	:=  iAdrMM2AmmBase;

	xMsg2354.Num		:=	2354;
	xMsg2354.AmmInAdr	:=  iAdrAmmBase2MM;
	xMsg2354.AmmOutAdr	:=  iAdrMM2AmmBase;

	xMsg2366.Num		:=	2366;
	xMsg2366.AmmInAdr	:=  iAdrAmmBase2MM;
	xMsg2366.AmmOutAdr	:=  iAdrMM2AmmBase;

	xMsg2688.Num		:=	2688;
	xMsg2688.AmmInAdr	:=  iAdrAmmBase2MM;
	xMsg2688.AmmOutAdr	:=  iAdrMM2AmmBase;

	xMsg2692.Num		:=	2692;
	xMsg2692.AmmInAdr	:=  iAdrAmmBase2MM;
	xMsg2692.AmmOutAdr	:=  iAdrMM2AmmBase;

	xMsg2693.Num		:=	2693;
	xMsg2693.AmmInAdr	:=  iAdrAmmBase2MM;
	xMsg2693.AmmOutAdr	:=  iAdrMM2AmmBase;

	xMsg2730.Num		:=	2730;
	xMsg2730.AmmInAdr	:=  iAdrAmmBase2MM;
	xMsg2730.AmmOutAdr	:=  iAdrMM2AmmBase;

	xMsg2801.Num		:=  2801;
	xMsg2801.AmmInAdr	:=  iAdrAmmBase2MM;
	xMsg2801.AmmOutAdr	:=  iAdrMM2AmmBase;

	xMsg2901.Num		:=  2901;
	xMsg2901.AmmInAdr	:=  iAdrAmmBase2MM;
	xMsg2901.AmmOutAdr	:=  iAdrMM2AmmBase;

	xMsg2902.Num		:=  2902;
	xMsg2902.AmmInAdr	:=  iAdrAmmBase2MM;
	xMsg2902.AmmOutAdr	:=  iAdrMM2AmmBase;

	xMsg2903.Num		:=  2903;
	xMsg2903.AmmInAdr	:=  iAdrAmmBase2MM;
	xMsg2903.AmmOutAdr	:=  iAdrMM2AmmBase;

	xMsg2934.Num		:=  2934;
	xMsg2934.AmmInAdr	:=  iAdrAmmBase2MM;
	xMsg2934.AmmOutAdr	:=  iAdrMM2AmmBase;

	xMsg3253.Num		:=  3253;
	xMsg3253.AmmInAdr	:=  iAdrAmmBase2MM;
	xMsg3253.AmmOutAdr	:=  iAdrMM2AmmBase;

	xMsg3254.Num		:=  3254;
	xMsg3254.AmmInAdr	:=  iAdrAmmBase2MM;
	xMsg3254.AmmOutAdr	:=  iAdrMM2AmmBase;

	xMsg3263.Num		:=  3263;
	xMsg3263.AmmInAdr	:=  iAdrAmmBase2MM;
	xMsg3263.AmmOutAdr	:=  iAdrMM2AmmBase;

	xMsg3264.Num		:=  3264;
	xMsg3264.AmmInAdr	:=  iAdrAmmBase2MM;
	xMsg3264.AmmOutAdr	:=  iAdrMM2AmmBase;

	xMsg3265.Num		:=  3265;
	xMsg3265.AmmInAdr	:=  iAdrAmmBase2MM;
	xMsg3265.AmmOutAdr	:=  iAdrMM2AmmBase;

	xMsg3266.Num		:=  3266;
	xMsg3266.AmmInAdr	:=  iAdrAmmBase2MM;
	xMsg3266.AmmOutAdr	:=  iAdrMM2AmmBase;

	xMsg3267.Num		:=  3267;
	xMsg3267.AmmInAdr	:=  iAdrAmmBase2MM;
	xMsg3267.AmmOutAdr	:=  iAdrMM2AmmBase;

	xMsg3269.Num		:=  3269;
	xMsg3269.AmmInAdr	:=  iAdrAmmBase2MM;
	xMsg3269.AmmOutAdr	:=  iAdrMM2AmmBase;

	xMsg3296.Num		:=  3296;
	xMsg3296.AmmInAdr	:=  iAdrAmmBase2MM;
	xMsg3296.AmmOutAdr	:=  iAdrMM2AmmBase;

	xMsg3297.Num		:=  3297;
	xMsg3297.AmmInAdr	:=  iAdrAmmBase2MM;
	xMsg3297.AmmOutAdr	:=  iAdrMM2AmmBase;

	xMsg3329.Num		:=  3329;
	xMsg3329.AmmInAdr	:=  iAdrAmmBase2MM;
	xMsg3329.AmmOutAdr	:=  iAdrMM2AmmBase;

	xMsg3352.Num		:=  3352;
	xMsg3352.AmmInAdr	:=  iAdrAmmBase2MM;
	xMsg3352.AmmOutAdr	:=  iAdrMM2AmmBase;

	xMsg3400.Num		:=  3400;
	xMsg3400.AmmInAdr	:=  iAdrAmmBase2MM;
	xMsg3400.AmmOutAdr	:=  iAdrMM2AmmBase;

	xMsg3412.Num		:=  3412;
	xMsg3412.AmmInAdr	:=  iAdrAmmBase2MM;
	xMsg3412.AmmOutAdr	:=  iAdrMM2AmmBase;

	xMsg3575.Num		:=  3575;
	xMsg3575.AmmInAdr	:=  iAdrAmmBase2MM;
	xMsg3575.AmmOutAdr	:=  iAdrMM2AmmBase;

	xMsg3576.Num		:=  3576;
	xMsg3576.AmmInAdr	:=  iAdrAmmBase2MM;
	xMsg3576.AmmOutAdr	:=  iAdrMM2AmmBase;

	xMsg3577.Num		:=  3577;
	xMsg3577.AmmInAdr	:=  iAdrAmmBase2MM;
	xMsg3577.AmmOutAdr	:=  iAdrMM2AmmBase;

	xMsg9244.Num		:=  9244;
	xMsg9244.AmmInAdr	:=  iAdrAmmBase2MM;
	xMsg9244.AmmOutAdr	:=  iAdrMM2AmmBase;

	xMsg9245.Num		:=  9245;
	xMsg9245.AmmInAdr	:=  iAdrAmmBase2MM;
	xMsg9245.AmmOutAdr	:=  iAdrMM2AmmBase;

	xMsg9304.Num		:=  9304;
	xMsg9304.AmmInAdr	:=  iAdrAmmBase2MM;
	xMsg9304.AmmOutAdr	:=  iAdrMM2AmmBase;

	xMsg9331.Num		:=  9331;
	xMsg9331.AmmInAdr	:=  iAdrAmmBase2MM;
	xMsg9331.AmmOutAdr	:=  iAdrMM2AmmBase;

	xMsg9083.Num		:=  9083;
	xMsg9083.AmmInAdr	:=  iAdrAmmBase2MM;
	xMsg9083.AmmOutAdr	:=  iAdrMM2AmmBase;

	xMsg9084.Num		:=  9084;
	xMsg9084.AmmInAdr	:=  iAdrAmmBase2MM;
	xMsg9084.AmmOutAdr	:=  iAdrMM2AmmBase;

	xMsg9085.Num		:=  9085;
	xMsg9085.AmmInAdr	:=  iAdrAmmBase2MM;
	xMsg9085.AmmOutAdr	:=  iAdrMM2AmmBase;

	xMsg9382.Num		:=  9382;
	xMsg9382.AmmInAdr	:=  iAdrAmmBase2MM;
	xMsg9382.AmmOutAdr	:=  iAdrMM2AmmBase;

	xMsg9383.Num		:=  9383;
	xMsg9383.AmmInAdr	:=  iAdrAmmBase2MM;
	xMsg9383.AmmOutAdr	:=  iAdrMM2AmmBase;

	(* template
	xMsg.Num		:=	;
	xMsg.AmmInAdr	:=  iAdrAmmBase2MM;
	xMsg.AmmOutAdr	:=  iAdrMM2AmmBase;
	*)
END_PROGRAM
```

#### MsgSY.var
```iecst
VAR
	iAdrAmmBase2MM : UDINT;
	iAdrMM2AmmBase : UDINT;
	xMsg1039 : Msg;
	xMsg1041 : Msg;
	xMsg1042 : Msg;
	xMsg1109 : Msg;
	xMsg1175 : Msg;
	xMsg1189 : Msg;
	xMsg1209 : Msg;
	xMsg1210 : Msg;
	xMsg1211 : Msg;
	xMsg1212 : Msg;
	xMsg1213 : Msg;
	xMsg1214 : Msg;
	xMsg1216 : Msg;
	xMsg1217 : Msg;
	xMsg1218 : Msg;
	xMsg1219 : Msg;
	xMsg1220 : Msg;
	xMsg1221 : Msg;
	xMsg1222 : Msg;
	xMsg1235 : Msg;
	xMsg1236 : Msg;
	xMsg2139 : Msg;
	xMsg2330 : Msg;
	xMsg2354 : Msg;
	xMsg2366 : Msg;
	xMsg2688 : Msg;
	xMsg2692 : Msg;
	xMsg2693 : Msg;
	xMsg2730 : Msg;
	xMsg2801 : Msg;
	xMsg2901 : Msg;
	xMsg2902 : Msg;
	xMsg2903 : Msg;
	xMsg2934 : Msg;
	xMsg3253 : Msg;
	xMsg3254 : Msg;
	xMsg3263 : Msg;
	xMsg3264 : Msg;
	xMsg3265 : Msg;
	xMsg3266 : Msg;
	xMsg3267 : Msg;
	xMsg3269 : Msg;
	xMsg3296 : Msg;
	xMsg3297 : Msg;
	xMsg3329 : Msg;
	xMsg3352 : Msg;
	xMsg3400 : Msg;
	xMsg3412 : Msg;
	xMsg3575 : Msg;
	xMsg3576 : Msg;
	xMsg3577 : Msg;
	xMsg9244 : Msg;
	xMsg9245 : Msg;
	xMsg9304 : Msg;
	xMsg9331 : Msg;
	xMsg9083 : Msg;
	xMsg9084 : Msg;
	xMsg9085 : Msg;
	xMsg9382 : Msg;
	xMsg9383 : Msg;
	ton_mcb_cf : TON;
	ctd_mcb_cf : CTD;
	ton_ctd_mcb : TON;
	ton_mcb_cf1 : TON;
	r_trig_mcb_ct : R_TRIG;
	r_trig_mcb_on : R_TRIG;
	ton_mcb_on : TON;
	ton_gcb_psf : TON;
	ton_gcb_opf : TON;
	r_trig_gcb_ct : R_TRIG;
	ton_ctd_gcb : TON;
	ctd_gcb_cf : CTD;
	r_trig_gcb_on : R_TRIG;
	ton_gcb_on : TON;
	ton_gcb_cf1 : TON;
	bN_EngStart1 : BOOL; (*engine start speed and 1 cycle*)
	xTON_SYST1 : TON;
	xTON_SYST2 : TON;
	xGR_MAX_LSA_LD : GR_MAXR;
	xTON_LSA_LD : TON;
	xTON_LSA : TON;
	xGR_MINR_P_Lo : GR_MINR;
	xGR_MAXR_P_Hi : GR_MAXR;
	xTON_P_Hi : TON; (*105%Pn 15s delay*)
	xTP_GCB_On : TP;
	xTOF_bGen2_Act : TOF;
	xGR_MAXR_P_Hi110 : GR_MAXR;
	xTON_P_Hi110 : TON; (*110%Pn 3s delay*)
	xTP_MMD_SynchDO : TP;
	xTON_P_HiHi : TON; (*120%Pn 500ms delay*)
	xGR_MAXR_P_HiHi : GR_MAXR;
	xTON_ParaInit_P_LimHiHi : TON;
	xTON_ParaInit_Ti_P_LimHiHi : TON;
	xTP_gcb_on : TP;
	xF_TRIG_gcb_on : F_TRIG;
	xR_TRIG_gcb_OnOffct : R_TRIG;
	xCTD_gcb_OnOffEvent : CTD;
	xTOF1216 : TOF;
	xTP_B9084 : TP; (*B9084 disappear after 20s*)
	xTON_gcb_psf_P_rev : TON; (*gcb position failure detected and reverse power 5s*)
END_VAR
```

### Program Logical/Synchronization/mains (IEC, version 4.13.0) - mains 

#### mainsCyclic.st
```iecst
(*******************************************************************************
mains 			mains ok detection for sy-control

This code is confidential and proprietary to the INNIO Company.
It may not be used in any form, or reproduced in any manner,
without the express written permission of the INNIO Company.
Copyright, INNIO Company, 2019

Customized modifications: -
------------------------

History:
-------
V1.10	12.01.2006	lettenb.	new
V1.11	16.03.2006	lettenb.	scb[1].on/off replaced with tie_on/off
V2.12	24.04.2006	LH			adapted for esy new
		11.11.2006	LH			revised after Para.bMSy test
V2.60.0	08.10.2009  lettenb.	ton_bb_dead: all_mcb_off     -> NOT any_mcb_on
										  	  all_gcb_off_bb -> NOT any_gcb_on_bb
								(->reset bb_dead with cb.on,
								hold gcb.command_on until cb=closed (gcb.aut_on2dead_bb))
V3.90.0	14.09.2011	lettenb.	Para.tiMainsOkDelay as parameter
V4.03.0	22.07.2015				OUT_SY.bRelMainsConnect new, dyn.gridcode III(thaler)
		25.07.2015  Plattner	OUT_SY.tMCB_COf_GCB_OpF.Do added, for opening MCB in CASE OF openingfailure GCB after set time in parameters
		30.09.2015  Plattner	OUT_SY.tParallel_Op.Do and OUT_SY.tIsland_Op.Do added for feedback
V4.04.0	22.07.2015	lettenb.	OUT_SY.tLockEng_ClosCond.Do new, bBB_ClosCond_Ok logic chnaged, dyn.gridcode III(thaler)
		07.10.2016				bBB_ClosCond_Ok logic changed acc.kiel validation
V4.05.0	28.12.2017	lettenb.	ssBusVoltPh -> tU_Bus_L, mapping cleanup
        03.01.2018              bBB_AfMnsF_ClosCond_Ok added, grid code logic(thaler)
		09.02.2018				bBBClosCond_Fault: xOpMode.NetP -> tGCB_On.Di(thaler)
V4.05.1 11.04.2018	lettenb.	trig_plc_on added, reset ton_mns_ok to avoid 1175 mains failure + 1189 at plc startup
V4.10.0 15.10.2020	lettenb.	ton_mns_ok: MIF only active, when island is not released, bugfix
V4.12.0 09.12.2022	lettenb.	bBBClosCond_Fault: closing conditions ignored when param.#14136 = FALSE, #921
V4.13.0	20.11.2023	Farre,		added IN_SY.bBypassMCB_deadBB interface from CU needed for Microgrid (2023-168)
		29.11.2023	Goenczi		bMainsReturn condition - take over Aggreko condition to standard

Instructions for use:
--------------------

Outstandings:
------------
locking first switch on all cb's
*******************************************************************************)
PROGRAM _CYCLIC

	IF	Para.bSyActive	THEN
		(*----------------------------------------------------------------------------*)
		(* busbar dead (OUT_SY.bBB_dead) *)
		xTON_BB_Dead(IN:= NOT bb_alive AND (IN_SY.bBypassMCB_deadBB OR NOT mcb.on) AND NOT any_gcb_on_bb, PT:= T#2s);
		bb_dead		:=	xTON_BB_Dead.Q;

		(*----------------------------------------------------------------------------*)
		(* micro interruption filter (KU-filter) *)
		tof_mns_ok(IN:=	mains.ok, PT:= Para.tiMIF);				(* micro interruption filter time *)

		(* mains return (OUT_SY.bMainsReturn) *)
		IF	Para.bMIF_Enable AND NOT IN_SY.tGCB_RI.Di THEN
			ton_mns_ok(IN := tof_mns_ok.Q, PT:= Para.tiMainsOkDelay);	(* micro interruption filter     active *)
		ELSE
			ton_mns_ok(IN := mains.ok,     PT:= Para.tiMainsOkDelay);	(* micro interruption filter not active *)
		END_IF;

		IF	ton_mns_ok.IN AND NOT ton_mns_ok.Q	THEN				(* countdown *)
			mains.return_rest_time := TIME_TO_DINT(ton_mns_ok.PT - ton_mns_ok.ET);
		ELSE
			mains.return_rest_time := 0;
		END_IF;

		trig_mcb_on(CLK:=	mcb.on);
		trig_sss_man(CLK:=	NOT	bSyOMSS_Aut);
		trig_plc_on(CLK:=   mains.ok AND IN_SY.tPB2MM.bSys_Run AND NOT IN_SY.tPB2MM.bParaSetupOk);(* reset at plc startup *)

		IF	trig_mcb_on.Q OR trig_sss_man.Q	OR trig_plc_on.Q THEN
			ton_mns_ok(IN:=	TRUE, PT:= T#0s); 		// PT_zero;		(* reset delay time *)
		END_IF;

		bMainsReturn	:=	ton_mns_ok.Q OR (mains.ok AND IN_SY.bSetFixedPwrMode AND IN_SY.tEng_Run.Do);

		(*----------------------------------------------------------------------------*)
		(* pulse mains ok (T_NE_OK) *)
		tp_p_mns_ok(IN:= ton_p_mns_ok.Q, PT:= T#100ms);
		ton_p_mns_ok(IN:= NOT mains.ok AND NOT tp_p_mns_ok.Q, PT:= T#2s);

		OUT_SY.tPulseMainsOk.Do :=  tp_p_mns_ok.Q;

		(*----------------------------------------------------------------------------*)
		(* synch line pulse *)
		ton_sy_line_of(IN:= (gcb.dmnd_sy OR mcb.dmnd_sy) AND NOT ton_sy_line_on.Q, PT:= T#120s);
		ton_sy_line_on(IN:= (gcb.dmnd_sy OR mcb.dmnd_sy) AND     ton_sy_line_of.Q, PT:= T#120s);

		pulse_sy_line	  := ton_sy_line_of.Q;

		(*----------------------------------------------------------------------------*)

	END_IF;

	(*----------------------------------------------------------------------------*)
	(* Closing conditions for busbar - GRID Code III *)
	(*----------------------------------------------------------------------------*)
	(* Boundary conditions for busbar - norm voltage and frequency *)
	IF 	    (IN_SY.tU_Bus_L1_2[1].Ai >= (Para.rU_BusNom[1]*(Para.rU_BB_ClosCond_LimLo_Norm + Para.rU_BB_ClosCond_Hy_Norm)))
		AND (IN_SY.tU_Bus_L2_3[1].Ai >= (Para.rU_BusNom[1]*(Para.rU_BB_ClosCond_LimLo_Norm + Para.rU_BB_ClosCond_Hy_Norm)))
		AND (IN_SY.tU_Bus_L3_1[1].Ai >= (Para.rU_BusNom[1]*(Para.rU_BB_ClosCond_LimLo_Norm + Para.rU_BB_ClosCond_Hy_Norm)))

		AND (IN_SY.tU_Bus_L1_2[1].Ai <= (Para.rU_BusNom[1]*(Para.rU_BB_ClosCond_LimHi_Norm - Para.rU_BB_ClosCond_Hy_Norm)))
		AND (IN_SY.tU_Bus_L2_3[1].Ai <= (Para.rU_BusNom[1]*(Para.rU_BB_ClosCond_LimHi_Norm - Para.rU_BB_ClosCond_Hy_Norm)))
		AND (IN_SY.tU_Bus_L3_1[1].Ai <= (Para.rU_BusNom[1]*(Para.rU_BB_ClosCond_LimHi_Norm - Para.rU_BB_ClosCond_Hy_Norm))) THEN

			bU_BB_ClosCond := TRUE;

	ELSIF  (IN_SY.tU_Bus_L1_2[1].Ai > (Para.rU_BusNom[1]*Para.rU_BB_ClosCond_LimHi_Norm))
		OR (IN_SY.tU_Bus_L2_3[1].Ai > (Para.rU_BusNom[1]*Para.rU_BB_ClosCond_LimHi_Norm))
		OR (IN_SY.tU_Bus_L3_1[1].Ai > (Para.rU_BusNom[1]*Para.rU_BB_ClosCond_LimHi_Norm))

		OR (IN_SY.tU_Bus_L1_2[1].Ai < (Para.rU_BusNom[1]*Para.rU_BB_ClosCond_LimLo_Norm))
		OR (IN_SY.tU_Bus_L2_3[1].Ai < (Para.rU_BusNom[1]*Para.rU_BB_ClosCond_LimLo_Norm))
		OR (IN_SY.tU_Bus_L3_1[1].Ai < (Para.rU_BusNom[1]*Para.rU_BB_ClosCond_LimLo_Norm)) THEN

			bU_BB_ClosCond := FALSE;

	END_IF;

	bBB_ClosCond_Ok := (IN_SY.tMnsOk_ClosCond_Ok.Di
			 	AND NOT(Para.bBB_ClosCondLimits_Active AND NOT IN_SY.tMnsOk_ClosCond_Skip.Di))
		    OR (       (Para.bBB_ClosCondLimits_Active AND NOT IN_SY.tMnsOk_ClosCond_Skip.Di)
				 	AND IN_SY.tMnsOk_ClosCond_Ok.Di
				 	AND bU_BB_ClosCond
				 	AND bF_BB_ClosCond);

	(* Boundary conditions for busbar after mains failure - norm voltage and frequency *)
	IF 	    (IN_SY.tU_Bus_L1_2[1].Ai >= (Para.rU_BusNom[1]*(Para.rU_BB_AfMnsF_ClosCond_LimLo_Norm + Para.rU_BB_AfMnsF_ClosCond_Hy_Norm)))
		AND (IN_SY.tU_Bus_L2_3[1].Ai >= (Para.rU_BusNom[1]*(Para.rU_BB_AfMnsF_ClosCond_LimLo_Norm + Para.rU_BB_AfMnsF_ClosCond_Hy_Norm)))
		AND (IN_SY.tU_Bus_L3_1[1].Ai >= (Para.rU_BusNom[1]*(Para.rU_BB_AfMnsF_ClosCond_LimLo_Norm + Para.rU_BB_AfMnsF_ClosCond_Hy_Norm)))

		AND (IN_SY.tU_Bus_L1_2[1].Ai <= (Para.rU_BusNom[1]*(Para.rU_BB_AfMnsF_ClosCond_LimHi_Norm - Para.rU_BB_AfMnsF_ClosCond_Hy_Norm)))
		AND (IN_SY.tU_Bus_L2_3[1].Ai <= (Para.rU_BusNom[1]*(Para.rU_BB_AfMnsF_ClosCond_LimHi_Norm - Para.rU_BB_AfMnsF_ClosCond_Hy_Norm)))
		AND (IN_SY.tU_Bus_L3_1[1].Ai <= (Para.rU_BusNom[1]*(Para.rU_BB_AfMnsF_ClosCond_LimHi_Norm - Para.rU_BB_AfMnsF_ClosCond_Hy_Norm))) THEN

			bU_BB_AfMnsF_ClosCond := TRUE;

	ELSIF  (IN_SY.tU_Bus_L1_2[1].Ai > (Para.rU_BusNom[1]*Para.rU_BB_AfMnsF_ClosCond_LimHi_Norm))
		OR (IN_SY.tU_Bus_L2_3[1].Ai > (Para.rU_BusNom[1]*Para.rU_BB_AfMnsF_ClosCond_LimHi_Norm))
		OR (IN_SY.tU_Bus_L3_1[1].Ai > (Para.rU_BusNom[1]*Para.rU_BB_AfMnsF_ClosCond_LimHi_Norm))

		OR (IN_SY.tU_Bus_L1_2[1].Ai < (Para.rU_BusNom[1]*Para.rU_BB_AfMnsF_ClosCond_LimLo_Norm))
		OR (IN_SY.tU_Bus_L2_3[1].Ai < (Para.rU_BusNom[1]*Para.rU_BB_AfMnsF_ClosCond_LimLo_Norm))
		OR (IN_SY.tU_Bus_L3_1[1].Ai < (Para.rU_BusNom[1]*Para.rU_BB_AfMnsF_ClosCond_LimLo_Norm)) THEN

			bU_BB_AfMnsF_ClosCond := FALSE;

	END_IF;

	bBB_AfMnsF_ClosCond_Ok :=  (IN_SY.tAfMnsF_ClosCond_Ok.Di
					 	AND NOT(Para.bBB_AfMnsF_ClosCondLimits_Active AND NOT IN_SY.tAfMnsF_ClosCond_Skip.Di))
				    OR (       (Para.bBB_AfMnsF_ClosCondLimits_Active AND NOT IN_SY.tAfMnsF_ClosCond_Skip.Di)
						 	AND IN_SY.tAfMnsF_ClosCond_Ok.Di
						 	AND bU_BB_AfMnsF_ClosCond
						 	AND bF_BB_AfMnsF_ClosCond);

	(*----------------------------------------------------------------------------*)
	(* Delay time conditions *)
	IF Para.bBB_AfMnsF_ClosCondLimits_Active THEN
		IF NOT IN_SY.tMnsOk.Di THEN
			bBBClosCond_Fault := TRUE;		(* status after mains failure ON *)
		ELSIF IN_SY.tGCB_On.Di THEN
			bBBClosCond_Fault := FALSE;		(* status after mains failure OFF *)
		END_IF;
	ELSE
		bBBClosCond_Fault := FALSE;
	END_IF;

	(* closing conditions mains ok (A) *)
	xTON_ClosCond(IN:= bBB_ClosCond_Ok, PT:= Para.tiBB_ClosCond_Delay);
	bAMM_ClosCond_Ok := xTON_ClosCond.Q;
	OUT_SY.tClosCond.Do	:= bAMM_ClosCond_Ok;

	(* closing conditions after mains failure (B) *)
	xTON_AfMnsF_ClosCond(IN:= bBB_AfMnsF_ClosCond_Ok, PT:= Para.tiBB_ClosCondAftMnsFail_Delay);
	bAMM_AfMnsF_ClosCond_Ok := xTON_AfMnsF_ClosCond.Q;
	OUT_SY.tAfMnsF_ClosCond.Do := bAMM_AfMnsF_ClosCond_Ok;

	OUT_SY.bRelMainsConnect	:= (NOT bBBClosCond_Fault AND bAMM_ClosCond_Ok)
							OR (	bBBClosCond_Fault AND bAMM_AfMnsF_ClosCond_Ok);

	(*----------------------------------------------------------------------------*)
	(* BEL Standard *)
	(* opens MCB in case of GCB opening failure *)
	xTON_MCB_COf_GCB_OpF(IN:= NOT IN_SY.tGCB_Off.Di AND IN_SY.tMCB_On.Di AND MM2VIS.bMsg1218, PT:= Para.tiMCB_COf_GCB_OpF);

	OUT_SY.tMCB_COf_GCB_OpF.Do 	:= xTON_MCB_COf_GCB_OpF.Q;
	(*----------------------------------------------------------------------------*)

	(*----------------------------------------------------------------------------*)
	(* BEL Standard *)
	(* Feedback mains parallel operation *)
	OUT_SY.tParallel_Op.Do := IN_SY.tMCB_On.Di AND IN_SY.tGCB_On.Di;

	(* Feedback Island operation *)
	OUT_SY.tIsland_Op.Do := NOT IN_SY.tMCB_On.Di AND IN_SY.tGCB_On.Di AND NOT IN_SY.bEng_Dem_EPS;

	(* Feedback emergency operation *)
	OUT_SY.tIsland_Op.Do := NOT IN_SY.tMCB_On.Di AND IN_SY.tGCB_On.Di AND IN_SY.bEng_Dem_EPS;
	(*----------------------------------------------------------------------------*)

END_PROGRAM
```

#### mains.var
```iecst
VAR
	xTON_BB_Dead : TON;
	tof_mns_ok : TOF;
	ton_sy_line_of : TON;
	ton_sy_line_on : TON;
	ton_p_mns_ok : TON;
	tp_p_mns_ok : TP;
	trig_sss_man : R_TRIG;
	trig_mcb_on : R_TRIG;
	ton_mns_ok : TON;
	bU_BB_ClosCond : BOOL; (* Closing condition buabar voltage *)
	bBB_ClosCond_Ok : BOOL; (* Delay time enabling *)
	xTON_ClosCond : TON; (* Timer for closing conditions delay time *)
	xTON_AfMnsF_ClosCond : TON; (* Timer for closing conditions delay time *)
	xTON_MCB_COf_GCB_OpF : TON;
	bU_BB_AfMnsF_ClosCond : BOOL;
	bBB_AfMnsF_ClosCond_Ok : BOOL;
	trig_plc_on : R_TRIG;
END_VAR
```

### Program Logical/Synchronization/mainsTC2 (IEC, version 4.05.0) - mains TC2

#### mainsTC2Cyclic.st
```iecst
(*******************************************************************************
mainsTC2 			mains

This code is confidential and proprietary to the INNIO Company.
It may not be used in any form, or reproduced in any manner,
without the express written permission of the INNIO Company.
Copyright, INNIO Company, 2019

Customized modifications: -
------------------------

History:
-------
V4.04.0	07.10.2016	lettenb.	new for fast detection of frequency changes, dyn.gridcode III(thaler)
V4.05.0	03.01.2018	lettenb.	bF_BB_AfMnsF_ClosCond added, grid code logic(thaler)
								IN_SY.tF_MMD_Synch2[1].Ai -> IN_SY.tF_MMD_BusBar[1].Ai

Instructions for use:
--------------------
IN_SY.tF_MMD_Synch2 mapping to Cyclic#2

Outstandings:
------------

*******************************************************************************)

PROGRAM _CYCLIC
 bF_BB_ClosCond_ZW_on  := FALSE;
 bF_BB_ClosCond_ZW_off := FALSE;

(* closing condition bus bar frequency *)
	IF 	   (IN_SY.tF_MMD_BusBar[1].Ai >= (Para.rF_BB_ClosCond_LimLo + Para.rF_BB_ClosCond_Hy))
		AND(IN_SY.tF_MMD_BusBar[1].Ai <= (Para.rF_BB_ClosCond_LimHi - Para.rF_BB_ClosCond_Hy)) THEN
		bF_BB_ClosCond_ZW_on  := TRUE;
	ELSIF  (IN_SY.tF_MMD_BusBar[1].Ai > Para.rF_BB_ClosCond_LimHi)
		OR (IN_SY.tF_MMD_BusBar[1].Ai < Para.rF_BB_ClosCond_LimLo) THEN
		bF_BB_ClosCond_ZW_off := TRUE;
	END_IF;

	(* Verzögerung für kurzen Wischer Messsignal *)
	xTON_F_BB_ClosCond_ZW_on (IN:= bF_BB_ClosCond_ZW_on,  PT:= T#1s);
	xTON_F_BB_ClosCond_ZW_off(IN:= bF_BB_ClosCond_ZW_off, PT:= T#80ms);

	IF    xTON_F_BB_ClosCond_ZW_on.Q THEN
		bF_BB_ClosCond := TRUE;
	ELSIF xTON_F_BB_ClosCond_ZW_off.Q THEN
		bF_BB_ClosCond := FALSE;
	END_IF;

(*-------------------------------------------------------------------------------------------------------------*)
 bF_BB_AfMnsF_ClosCond_ZW_on  := FALSE;
 bF_BB_AfMnsF_ClosCond_ZW_off := FALSE;

(* closing condition bus bar frequency - after mains failure *)
	IF 	   (IN_SY.tF_MMD_BusBar[1].Ai >= (Para.rF_BB_AfMnsF_ClosCond_LimLo + Para.rF_BB_AfMnsF_ClosCond_Hy))
		AND(IN_SY.tF_MMD_BusBar[1].Ai <= (Para.rF_BB_AfMnsF_ClosCond_LimHi - Para.rF_BB_AfMnsF_ClosCond_Hy)) THEN
		bF_BB_AfMnsF_ClosCond_ZW_on  := TRUE;
	ELSIF  (IN_SY.tF_MMD_BusBar[1].Ai > Para.rF_BB_AfMnsF_ClosCond_LimHi)
		OR (IN_SY.tF_MMD_BusBar[1].Ai < Para.rF_BB_AfMnsF_ClosCond_LimLo) THEN
		bF_BB_AfMnsF_ClosCond_ZW_off := TRUE;
	END_IF;

	(* Verzögerung für kurzen Wischer Messsignal *)
	xTON_F_BB_AfMnsF_ClosCond_ZW_on (IN:= bF_BB_AfMnsF_ClosCond_ZW_on,  PT:= T#1s);
	xTON_F_BB_AfMnsF_ClosCond_ZW_off(IN:= bF_BB_AfMnsF_ClosCond_ZW_off, PT:= T#80ms);

	IF    xTON_F_BB_AfMnsF_ClosCond_ZW_on.Q THEN
		bF_BB_AfMnsF_ClosCond := TRUE;
	ELSIF xTON_F_BB_AfMnsF_ClosCond_ZW_off.Q THEN
		bF_BB_AfMnsF_ClosCond := FALSE;
	END_IF;

END_PROGRAM
```

#### mainsTC2Init.st
```iecst
(********************************************************************
 * COPYRIGHT -- INNIO Company
 ********************************************************************
 * Program: mainsf
 * File: mainsfInit.st
 * Author: 105035758
 * Created: August 24, 2016
 ********************************************************************
 * Implementation of program mainsf
 ********************************************************************)

PROGRAM _INIT

(* TODO : Add your code here *)

END_PROGRAM
```

#### mainsTC2.var
```iecst
VAR
	bF_BB_ClosCond_ZW_on : BOOL := 0;
	bF_BB_ClosCond_ZW_off : BOOL := 0;
	xTON_F_BB_ClosCond_ZW_on : TON;
	xTON_F_BB_ClosCond_ZW_off : TON;

	bF_BB_AfMnsF_ClosCond_ZW_on : BOOL := 0;
	bF_BB_AfMnsF_ClosCond_ZW_off : BOOL := 0;
	xTON_F_BB_AfMnsF_ClosCond_ZW_on : TON;
	xTON_F_BB_AfMnsF_ClosCond_ZW_off : TON;
END_VAR
```

### Program Logical/Synchronization/gcb (IEC, version 4.13.0) - generator circuit breaker control

#### gcbCyclic.st
```iecst
(*******************************************************************************
gcb 		generator circuit breaker control

This code is confidential and proprietary to the INNIO Company.
It may not be used in any form, or reproduced in any manner,
without the express written permission of the INNIO Company.
Copyright, INNIO Company, 2020

Customized modifications: -
------------------------

History:
-------
V1.10	12-01-2006	lettenb.	new
V1.11	16-03-2006	lettenb.	scb[1].on/off replaced with tie_on/off
V2.12	24.04.2006				LH	mcb1 imported from MSY
								mcb1 --> gcb
								adapted for esy new
		22.09.2006	LH			extented release gcb
		11.11.2006	LH			revised after Para.bMSy test
		20.11.2006	LH			revised for final release esy new
V2.20	07.02.2007	LH			-bridging gcb ready signal while winding up spring
								-demand synchronization: gcb.alarm --> gcb.monitoring_release
								-gcb on to dead busbar: alarm_voltage_sensor_bb1 integrated
								-advanced software documentation
V2.201	12.09.2007	LH			correction of network comments (FG_GSUW)
V2.30	18.01.2008	LH			adapted for test-bench run
		28.03.2008	LH			lock gcb in case of any position failure on busbar
V2.34.0	28.10.2008	lettenb.	Para.bBS_Acc_Active added
V2.50.0 28.01.2009	lettenb.	calm: IN_SY.bGCB_Off_RP, IN_SY.bGCB_Off_CNS added
V2.50.3 08.10.2009	lettenb.	tof_gcb_command_on added (extend gcb command on signal)
		30.11.2009  lettenb.	gcb.dmnd_sy:  n > 1400min-1 added
								(360min-1 + ton10"=IN_SY.tEng_Run.Do: ist zu früh!bei schlechter motoreinstellung
								 od. schlechter gasqualität)
V3.20.0	07.12.2010	lettenb.	P10proz added, selbsthaltung limit 10%Pnenn unterschritten wenn keine anford.
								(flackerndes limit setzt und löscht immer wieder on/off-command gcb (OUT_SY.tGCB_Cof.Do!))
V3.30.0	04.11.2011	lettenb.	gcb.release: IN_SY.tGCB_RGC.Do added
V3.90.0	25.10.2012	lettenb.	Para.bGridCode_Active added
V3.99.0 24.06.2013	lettenb.	tof_gcb_man_off: only active with NOT bSyOMSS_Aut
								(to avoid gcb opening at SyOMSS_Aut->Man, within 6" after pressed gcb.man_off)
								xGR_MAXR_P_HiNoManOff: Gw: 50.0 -> 0.5, bugfix
		23.06.2015	Graus,		type 6 load rejection - open gcb at full load
V4.03.0	29.07.2015	lettenb.	ton_gcb_dmnd_sy.PT := T#5s; removed(standardisierung für schnellstart/greenfrog)
                    plattner    temperature MAX generator switch gear power reduction and set,
V4.04.0	22.09.2016	lettenb.	Para.rP_Red_TempMax_GenCB_Rate   /100 removed and logic changed, bugfix
		11.10.2016	Perktold, 	Para.bGridCode_Active replaced by IN_SY.bGridCode_ON
		13.09.2018	lettenb.	ton_EINPF_2 moved for sequential arrangement, bu01
V4.07.0	17.12.2018	lettenb.	ton_gcb_dmnd_sy.IN: bGnlTrip added to avoid B2139"request synchr.",after gcb-opening by external protection(caused by removal of ton_gcb_dmnd_sy.PT), bugfix
V4.10.0	16.10.2020	Weitzer		IN_SY.bCust_Dem_Sy added to GCB demand sy
					lettenb.	GCB_OnCnt added
V4.11.0	24.06.2021	Arnold		Open GCB in island on underfrequency IN_SY.bGCB_DCon_EC
V4.12.0	07.12.2022	lettenb.	ton_gcb_dmnd_sy.PT: T#0s -> 100ms, to avoid B2139 caused by time overlap,#890
								OUT_SY.bGCB_aut_on2dead_bb added,#912
								ton_gcb_dmnd_sy.IN: bOMSS_Man removed(as validated with saarbrücken AA46/wasserer)
V4.13.0	17.08.2023	lettenb.	dead bb synch, bugfixes(BR21/wasserer,schwab,lettenb.)
		29.11.2023	Goenczi		GCB demand synch conditions extended to command from BUS

Instructions FOR use:
--------------------
task have to be operated after MsgSY

Outstandings:
------------
remove ton_gcb_dmnd_sy
*******************************************************************************)
PROGRAM _CYCLIC

	IF	Para.bSyActive	THEN
		(*----------------------------------------------------------------------------*)
		(* gcb demand synchronization (OUT_SY.bGCB_DemSy) *)
		gcb_dmnd_IN1 :=  	(   bSyOMSS_Aut             AND (NOT IN_SY.bBus_Active OR NOT IN_SY.bOM_Bus));	(*gcb auto on command *)
		gcb_dmnd_IN2 :=		   (IN_SY.bSetAutControlMode AND     IN_SY.bOM_Bus AND NOT IN_SY.bSetGCB2Open);		(*gcb auto on command from bus*)
		gcb_dmnd_IN3 :=   	   (bSyOMSS_Man									(* gcb manual on command *)
							AND		bOMSS_Man
							AND	NOT gcb.man_off
							AND	   (gcb.man_on OR ANW_ENTR OR ton_gcb_dmnd_sy.IN));
		gcb_dmnd_IN4 :=      (IN_SY.bOM_Bus 								(* gcb manual on command from bus *)
							AND NOT IN_SY.bSetAutControlMode
							AND     IN_SY.bSetManControlMode
							AND NOT IN_SY.bSetGCB2Open
							AND    (IN_SY.bSetGCB2Close OR ANW_ENTR OR ton_gcb_dmnd_sy.IN))  ;

		ton_gcb_dmnd_sy.IN :=  (gcb_dmnd_IN1 OR gcb_dmnd_IN2 OR gcb_dmnd_IN3 OR gcb_dmnd_IN4  )  	(* synchronization selected *)
					AND    (IN_SY.rN_EngAct > (Para.rN_EngNom * 0.933))  		(* n > 1400 *)
					AND		IN_SY.tRel_Sync_Load.Do								(* engine ready for load (IN_SY.tRel_Sync_Load.Do) *)
					AND		gcb.eng_demanded									(* engine demanded (IN_SY.bEng_RPSDem) *)
					AND 	gcb.rdy												(* gcb ready for closing *)
					AND NOT gcb.on												(* gcb is open *)
					AND 	gcb.mon_release										(* monitoring release gcb *)
					AND NOT	mcb.dmnd_sy											(* no mcb demand synchronization (OUT_SY.bMCB_DemSy) *)
					AND	NOT	mcb_man_on2dead_bb									(* no manual closing mcb1 to dead busbar *)
					AND	NOT	mcb_aut_on2dead_bb									(* no automatic closing mcb1 to dead busbar *)
					AND NOT	any_gcb_edc_bb										(* no lock from external unit *)
					AND	NOT	gcb.mdl												(* no lock from Para.bMSy *)
					AND	NOT	bGen_DeExc_Err										(* no de-excitation failure *)
					AND    (IN_SY.tGrC_DCon.Do OR NOT IN_SY.bGridCode_ON)		(* gridcode release (LVRT) *)
					AND NOT bGnlTrip
	 				AND		IN_SY.bCust_Dem_Sy									(* release by customer - external synchronisation *)
					AND		TRUE;												(* include additional release conditions *)

		ton_gcb_dmnd_sy.PT := T#100ms;
		ton_gcb_dmnd_sy();

		gcb.dmnd_sy	:=	ton_gcb_dmnd_sy.Q;										(* demand synchronization (OUT_SY.bGCB_DemSy) *)

		(*----------------------------------------------------------------------------*)
		(* release trip gcb *)
		ton_gcb_rel_trip(IN:= bDem_Island AND gcb.eng_oper, PT:= T#1s);

		gcb.rel_trip :=	ton_gcb_rel_trip.Q;										(* release trip gcb in case of mains failure *)

		(*----------------------------------------------------------------------------*)
		(* monitoring release gcb (FG_GSUW) *)
		gcb.mon_release :=	NOT gcb.alm_0sf										(* 0-signal failure gcb *)
						AND NOT gcb.alm_1sf										(* 1-signal failure gcb *)
						AND NOT gcb.alm_cf										(* closing failure gcb *)
						AND NOT any_gcb_opf_bb									(* gcb with opening failure *)
						AND NOT any_gcb_psf_bb									(* gcb with position failure *)
						AND	NOT	mcb.alm_opf										(* mains cb with opening failure *)
						AND	NOT	mcb.alm_psf										(* mains cb with position failure *)
						AND		mcb.remote										(* all mcb remote *)
						AND		IN_SY.tPB2MM.bSys_Run;							(* PLC running *)

		(*----------------------------------------------------------------------------*)
		(* release gcb *)
		ton_EINPF_1(IN:= NOT gcb.release             AND NOT IN_SY.tGCB_SM1.Di, PT:= T#5s);(* output signal test *)

		bSM1TestOk		:=	gcb.release
					OR	   (gcb.dmnd_sy AND ton_EINPF_1.Q);						(* digital output signal test ok *)
		(*-------------------------------------------------------------*)

		sy_lfg			:=	ton_EINPF_2.Q										(* relais contact signal test *)
					OR	   (sy_lfg AND IN_SY.tRel_Sync_Load.Do);

		ton_EINPF_2(IN:= NOT IN_SY.tRel_Sync_Load.Do AND     IN_SY.tGCB_SM2.Di, PT:= T#5s);(* relais contact signal test, this line have to be situated after building of sy_lfg! *)

		bSM2TestOk		:= (sy_lfg AND OUT_SY.tGCB_RUC.Do)						(* relais contact signal test ok *)
					OR		SY_LFG_THJ;

		SY_LFG_THJ		:=	sy_lfg;												(* extended load release (1 cycle) *)
		(*-------------------------------------------------------------*)

		bMnsConnection 	:=  mcb.on AND mains.ok AND	NOT	MM2VIS.bMsg3412;		(* mains connection ok *)

		NWK_RS			:=	Para.bMCB_ReSw2Mns_Enable
					AND	NOT	mcb.on												(* mcb open *)
					AND		bMainsReturn;										(* mains return (OUT_SY.bMainsReturn(1)) *)

		bRS2Mains		:=	NWK_RS												(* mains ok for reswitch to mains for customer *)
					AND		IN_SY.tGCB_DRM.Di;									(* release for reswitch to mains from customer *)

		gcb.release		:=	gcb.mon_release										(* monitoring release gcb  *)
					AND		bSM1TestOk											(* digital output signal test ok *)
					AND		bSM2TestOk											(* relais contact signal test ok *)
					AND    (gcb.rdy        OR gcb.on)							(* gcb ready for closing *)
					AND	   (bMnsConnection OR gcb.rel_trip) 					(* no decoupling from mains *)
					AND	NOT	bRS2Mains											(* no reswitch to mains *)
					AND	NOT	any_gcb_edc_bb										(* no lock from customer *)
					AND	NOT	gcb.mdl												(* no lock from Para.bMSy *)
					AND	NOT	IN_SY.bGCB_Off_RP									(* gcb off by gen.reverse power *)
					AND	NOT	IN_SY.bGCB_Off_CNS									(* gcb off by asym.current *)
					AND    (IN_SY.tGrC_DCon.Do OR NOT IN_SY.bGridCode_ON)		(* LVRT failure *)
					AND	NOT IN_SY.bGCB_DCon_EC									(* GCB open command from EngineController *)
					AND		TRUE;												(* include additional release conditions *)

		(*----------------------------------------------------------------------------*)
		tof_gcb_man_off(IN:= gcb.man_off AND bOMSS_Man AND NOT bSyOMSS_Aut, PT:= T#6s);	(* extended manual off command gcb *)
		tof_gcb_dmnd_sy(IN:= gcb.dmnd_sy, PT:= T#100ms);						(* extended demand synchronize gcb *)

		(*----------------------------------------------------------------------------*)
		(* gcb on to dead busbar (GS_AES/GS_1) *)
		gcb.aut_on2dead_bb := (bSyOMSS_Aut OR bSyOMSS_Man)						(* synchronization is active *)
					AND 	gcb.release											(* release gcb *)
					AND 	gcb.dmnd_sy											(* gcb demand synchronization (OUT_SY.bGCB_DemSy) *)
					AND( 	bb_dead	OR(IN_SY.tDemGenExcOff.Di AND NOT bb_alive))(* dead busbar (OUT_SY.bBB_dead) *)
					AND(NOT	MM2VIS.bMsg1216 OR	OUT_SY.bTestBenchModeIsland)	(* no busbar voltage sensor failure *)
					AND	NOT	any_gcb_psf_bb										(* no gcb with position failure *)
					AND(NOT	mcb.alm_psf OR OUT_SY.bTestBenchModeIsland)			(* no mains cb with position failure *)
					AND 	gcb.edc												(* demand closing gcb to dead busbar *)
					AND		rel_gcb_on2d_bb										(* release closing gcb to dead busbar *)
					AND		rel_load_shedd										(* load shedding ok *)
					AND	   (bGen_DeExc_Rdy OR NOT Para.bGenDeexit_Enable);		(* generator de-excited *)

		OUT_SY.bGCB_aut_on2dead_bb := gcb.aut_on2dead_bb;

		(*----------------------------------------------------------------------------*)
		(* release sy-puls gcb (SY) *)
		gcb.rel_sy_puls :=	gcb.release
					AND		tof_gcb_dmnd_sy.Q									(* extended demand synchronize gcb (T74) *)
					AND	   (bSyOMSS_Aut	OR (bSyOMSS_Man AND	NOT	tof_gcb_man_off.Q))
					AND NOT IN_SY.tDemGenExcOff.Di
					AND     bb_alive;

		(*----------------------------------------------------------------------------*)
		(* command gcb off *)
		bP_Lo_Hold		:=  (gcb.eng_demanded OR  bP_Lo_Hold) AND NOT bP_Lo;	(* hold P_Lo in case of flickering signal*)
		xGR_MAXR_P_HiNoManOff(In:= IN_SY.rP_Act_Norm_Filt, Gw:= 0.5, Hy:= 0.0); (* lockout manual gcb off command *)
																				(* with bOMSS_Aut + SyOMS_MAN: gcb can not be opened manually -> general topic *)
		gcb.dmnd_off 	:=	NOT gcb.release
						OR 	   (bOMSS_Man	AND		tof_gcb_man_off.Q	AND (NOT	xGR_MAXR_P_HiNoManOff.Q OR (Para.bP_LoadReject_Active AND IN_SY.bType6_Update_Rel)))
					    OR     (bOMSS_Aut	AND NOT gcb.eng_demanded 	AND(	NOT gcb.on
																			OR	NOT	bP_Lo_Hold
																			OR (NOT OUT_SY.bOtherGenParallel AND NOT mcb.on)))
					    OR     (bOMSS_Test	AND NOT gcb.eng_demanded 	AND(	NOT gcb.on
																			OR	NOT	bP_Lo_Hold
																			OR (NOT OUT_SY.bOtherGenParallel AND NOT mcb.on)))
						OR     (IN_SY.bOM_Bus AND IN_SY.bSetGCB2Open);			(*demand off from bus - Aggreko*)

		gcb.command_off :=	gcb.dmnd_off OR NOT IN_SY.tPB2MM.bSys_Run;			(* true = command off *)

		(*----------------------------------------------------------------------------*)
		(* command gcb on to dead busbar *)
		gcb.dmnd_on	:=	gcb.aut_on2dead_bb;

		tof_gcb_command_on(IN:= gcb.dmnd_on	AND	NOT	gcb.on AND NOT gcb.command_off AND IN_SY.tPB2MM.bSys_Run, PT:= T#100ms);

		gcb.command_on:= tof_gcb_command_on.Q;

		(*----------------------------------------------------------------------------*)

	END_IF;

	(* added from pb10 *)
	(*----------------------------------------------------------------------------*)
	(* Collective alarm Prio. 1 -> Switch OFF OUT_SY.tGCB_RUC.Do with new motor Off strategy *)
	xTP_GnlTrip1(IN:= bGnlTrip1, PT:= T#5s);

	(* gcb release under voltage coil *)
	OUT_SY.tGCB_RUC.Do := 	NOT IN_SY.bMsg1038 									(* generator reverse power	*)
						AND(NOT IN_SY.bMsg1026	OR IN_SY.bMsg1026_Test)			(* shutdown failure			*)
						AND(NOT MM2VIS.bMsg1041	OR       bMsg1041_Test)			(* power signal missing		*)
						AND(NOT MM2VIS.bMsg1042 OR       bMsg1042_Test)			(* power signal overload	*)
						AND NOT MM2VIS.bMsg1217									(* gcb status signal failure*)
						AND NOT MM2VIS.bMsg1219									(* gcb closing failure		*)
						AND NOT xTP_GnlTrip1.Q;

	(*----------------------------------------------------------------------------*)
	(* Temperature max generator switch gear (Power reduction) *)
	IF Para.bP_Red_TempMax_GenCB_Active AND NOT IN_SY.tTempMax_GenCB.Di THEN
		OUT_SY.bP_Red_TempMax_GenCB_Sel	:= TRUE;
		OUT_SY.rP_Red_TempMax_GenCB_Norm := LIMIT(0.5, Para.rP_Red_TempMax_GenCB_Rate, 1.0);
	ELSE(* Temperature max generator switch gear (Power reduction) inaktive*)
		OUT_SY.bP_Red_TempMax_GenCB_Sel	:= FALSE;
		OUT_SY.rP_Red_TempMax_GenCB_Norm := 1.0;
	END_IF;

	(*----------------------------------------------------------------------------*)
	(* gcb on counter *)
	IF EDGEPOS(gcb.on) THEN
		VIS2MM.iGCB_OnCnt := (VIS2MM.iGCB_OnCnt + 1) MOD 100000;	(* counter, check limits *)
	END_IF;

	(*----------------------------------------------------------------------------*)

END_PROGRAM
```

#### gcb.var
```iecst
VAR
	bSM1TestOk : BOOL;
	bSM2TestOk : BOOL;
	tof_gcb_man_off : TOF;
	tof_gcb_dmnd_sy : TOF;
	ton_gcb_rel_trip : TON;
	ton_EINPF_1 : TON;
	ton_EINPF_2 : TON;
	tof_gcb_command_on : TOF;
	bP_Lo_Hold : BOOL := FALSE;
	sy_lfg : BOOL;
	SY_LFG_THJ : BOOL;
	NWK_RS : BOOL; (*mains back for reswitch to mains for customer*)
	bRS2Mains : BOOL; (*reswitch to mains*)
	bMnsConnection : BOOL; (*mains connection ok*)
	xTP_GnlTrip1 : TP;
	xGR_MAXR_P_HiNoManOff : GR_MAXR;
	gcb_dmnd_IN1 : BOOL := 0; (*GCB demand auto*)
	gcb_dmnd_IN2 : BOOL := 0; (*GCB demand auto via bus coupling*)
	gcb_dmnd_IN3 : BOOL := 0; (*GCB demand manual*)
	gcb_dmnd_IN4 : BOOL := 0; (*GCB demand manual via bus coupling*)
END_VAR
```

### Program Logical/Synchronization/gcbTC1 (IEC, version 4.14.0) - generator circuit breaker TC1

#### gcbTC1Cyclic.st
```iecst
(*******************************************************************************
gcbTC1 		generator circuit breaker monitoring

This code is confidential and proprietary to the INNIO Company.
It may not be used in any form, or reproduced in any manner,
without the express written permission of the INNIO Company.
Copyright, INNIO Company, 2021

Customized modifications: -
------------------------

History:
-------
V4.09.0	11.09.2019	lettenb.	new
		30.01.2020	lettenb.	bResetWarning from general_SY, added, JMAP cleanup
		11.04.2020	lettenb.	current limit 10 -> 2% I_GenNom, testbench validation
V4.11.0 05.11.2021	lettenb.	hold last value with reset, bugfix
V4.14.0 22.11.2024	Fahringer	Use generator current before GCB closure to check 2% change (2024-238)
								GCB closing time monitoring for more than 40ms (2024-238)
		22.11.2024	Farre		bMMD_SyncDO only when used for GCB (2024-238)

Instructions FOR use:
--------------------
task have to be operated in 1ms task class

Outstandings:
------------
*******************************************************************************)
PROGRAM _CYCLIC

IF Para.bMMDSynch_Act[1] AND IN_SY.tPB2MM.bParaSetupOk THEN

	(* sy-pulse = start measurement *)
	xTP_MMD_SynchDO(IN:= IN_SY.bMMD_SynchDO_TC1[1], PT:= REAL_TO_TIME(rGCB_On_TimeMax));

	(* read phase current and GCB On status when Synch pulse is detected *)
	IF EDGEPOS(IN_SY.bMMD_SynchDO_TC1[1]) THEN
		rI_L1_bSync 	:= 	IN_SY.tI_L1_TC1[1].Unfilt;
		rI_L2_bSync 	:= 	IN_SY.tI_L2_TC1[1].Unfilt;
		rI_L3_bSync 	:= 	IN_SY.tI_L3_TC1[1].Unfilt;
		bGCB_On_bSync	:=	IN_SY.tGCB_On.Di;
	END_IF;

	(* start counter when synch pulse is detected *)
	IF xTP_MMD_SynchDO.Q THEN rCnt := rCnt + 1;
	                     ELSE rCnt := 0;
	END_IF;
	IF rCnt > 100000 THEN rCnt := 0;
	END_IF;

	(* gcb closed detection *)
	IF xTP_MMD_SynchDO.Q AND NOT bGCB_On_bSync THEN
		IF 	(ABS(IN_SY.tI_L1_TC1[1].Unfilt - rI_L1_bSync) > (Para.rI_GenNom[1] * 0.02)) OR
		 	(ABS(IN_SY.tI_L2_TC1[1].Unfilt - rI_L2_bSync) > (Para.rI_GenNom[1] * 0.02)) OR
			(ABS(IN_SY.tI_L3_TC1[1].Unfilt - rI_L3_bSync) > (Para.rI_GenNom[1] * 0.02))
		THEN
			bGCB_OnI := TRUE; (* hold status *)
		END_IF;
	ELSE
		bGCB_OnI := FALSE;
	END_IF;

	xR_TRIG_GCB_OnI(CLK:= (rCnt >=40) AND bGCB_OnI);
	xR_TRIG_Timeout(CLK:= (rCnt = rGCB_On_TimeMax) AND NOT bGCB_OnI);
	IF NOT bGCB_On_bSync AND (xR_TRIG_GCB_OnI.Q OR xR_TRIG_Timeout.Q) THEN
		rGCBctOld := rGCBct;
		rGCBct    := rCnt; (* ms *)
	END_IF;

	(* failure detection *)
	IF ((ABS(Para.rTi_SynchSwitchDel[1] - rGCBct   ) >= 20) AND (rCnt >=40))
		AND(ABS(Para.rTi_SynchSwitchDel[1] - rGCBctOld) >= 20)	THEN bGCBctd := TRUE; (* GCB closing time deviation *)
	END_IF;

	(* reset *)
	IF bGCBctd AND bResetWarning THEN
		bGCBctd   := FALSE;
		rGCBctOld := Para.rTi_SynchSwitchDel[1];
	END_IF;

	(* MM2VIS *)
	MM2VIS.tiGCB_ClosTime    := REAL_TO_TIME(rGCBct);
	MM2VIS.tiGCB_ClosTimeOld := REAL_TO_TIME(rGCBctOld);

ELSE

	bGCBctd := FALSE;
	rGCBctOld := Para.rTi_SynchSwitchDel[1];
	rGCBct    := Para.rTi_SynchSwitchDel[1];

	(* MM2VIS *)
	MM2VIS.tiGCB_ClosTime    := REAL_TO_TIME(rGCBct);
	MM2VIS.tiGCB_ClosTimeOld := REAL_TO_TIME(rGCBctOld);

END_IF;

END_PROGRAM
```

#### gcbTC1Init.st
```iecst
PROGRAM _INIT

	rGCBctOld := Para.rTi_SynchSwitchDel[1];
	rGCBct    := Para.rTi_SynchSwitchDel[1];
	bGCBctd   := FALSE;
	rGCB_On_TimeMax := 300; (* ms *)(* maximum measurement time 300+500=800ms !? *)

END_PROGRAM
```

#### gcbTC1.var
```iecst
VAR
	xR_TRIG_GCB_OnI : R_TRIG; (*positive edge detection GCB on pulse*)
	xR_TRIG_Timeout : R_TRIG; (*positive edge detection timout*)
	bGCB_OnI : BOOL; (*GCB On impulse detection*)
	rGCBct : REAL; (*gcb closing time*)
	rGCBctOld : REAL; (*gcb closing time one before last*)
	rGCB_On_TimeMax : REAL; (*Maximum time GCB On monitoring*)
	rCnt : REAL; (*GCB Closing time counter*)
	xTP_MMD_SynchDO : TP; (*MMU Pulse TP timer*)
	rI_L1_bSync : REAL := 0.0; (*Phase current L1 before synch pulse*)
	rI_L2_bSync : REAL := 0.0; (*Phase current L2 before synch pulse*)
	rI_L3_bSync : REAL := 0.0; (*Phase current L3 before synch pulse*)
	bGCB_On_bSync : BOOL := 0; (*GCB On status before synch pulse*)
END_VAR
```

### Program Logical/Synchronization/mcb (IEC, version 4.13.0) - mains circuit breaker control

#### mcbCyclic.st
```iecst
(*******************************************************************************
mcb				mains circuit breaker control

This code is confidential and proprietary to the INNIO Company.
It may not be used in any form, or reproduced in any manner,
without the express written permission of the INNIO Company.
Copyright, INNIO Company, 2022

Customized modifications: -
------------------------

History:
-------
V1.10	12.01.2006	lettenb.	new
V1.11	16.03.2006	lettenb.	scb[1].on/off replaced with tie_on/off
V2.12	24.04.2006	LH			adapted for esy new
		11.11.2006	LH			revised after Para.bMSy test
		20.11.2006	LH			revised for final release esy new
V2.20	07.02.2007	LH			adapted for supporting customer mcb
		27.04.2007	LH			update according to changes Para.bMSy:
								-mcb[x].command_on: tof_mcb_man_off[x].Q was mcb[x].command_off
								-ton_mcb_mrc[x] added
V2.60.0 13.08.2009	lettenb.	any_gcb_opf_bb changed by gcb[0].alm_opf, gcb_opf_delay
V3.30.0	10.10.2011	lettenb.	ton_mcb_dmnd_sy[1].IN: mcb.rdy added
V3.99.0	27.02.2013	lettenb.	cleanup
V4.09.0 05.02.2020	lettenb.	mcb[1].release_trip ruhestrom -> arbeitsstrom for mcb contr.by cust, missing change from V3.40.0 added
		20.04.2020	lettenb.	ton_mcb_dmnd_sy.IN:	mcb controlled by customer, bugfix(heim, Referenzanlage AB85)
		01.10.2020	lettenb.	ton_mcb_dmnd_sy.IN:	mcb controlled by customer, MCB_DVS also with bSyOMSS_Man, bu
V4.10.0	16.10.2020	Weitzer		mcb.man_on commented, IN_SY.bCust_Dem_RSy from CU added to ton_mcb_dmnd_sy ELSE part
V4.12.0 29.06.2022	lettenb.	dead bb synch added

Instructions for use:
--------------------

Outstandings:
------------
release mcb1 (old hardware design) to delete after testing
*******************************************************************************)
PROGRAM _CYCLIC

	IF	Para.bSyActive	THEN
		(*----------------------------------------------------------------------------*)
		(* mcb demand synchronization (OUT_SY.bMCB_DemSy) *)
		IF Para.bMCB_Enable THEN										(* mcb controlled by esy *)
			ton_mcb_dmnd_sy.IN :=  (bSyOMSS_Aut
								OR (bSyOMSS_Man AND	NOT	mcb.man_off AND (mcb.man_on OR ton_mcb_dmnd_sy.IN)))
							AND		mcb.remote
							AND	   (bSyOMSS_Man OR bMainsReturn)
							AND    (mains.ok    OR bMainsReturn)
							AND		mcb.release
							AND	NOT mcb.alarm

							AND 	mcb.rdy
							AND	NOT mcb.on
							AND	   (bb_alive OR any_eng_oper_and_gcb_on_bb)
							AND	NOT	Para.bMCB_ReSw2Mns_Enable
							AND	NOT	MM2VIS.bMsg3412;

		ELSE															(* mcb controlled by customer *)
			ton_mcb_dmnd_sy.IN :=  (bSyOMSS_Man OR bSyOMSS_Aut)
							AND		bMainsReturn
							AND	NOT	gcb.dmnd_sy

							AND 	mcb.rdy
							AND	NOT mcb.on
							AND	   (bb_alive OR any_eng_oper_and_gcb_on_bb)
							AND	NOT	Para.bMCB_ReSw2Mns_Enable
							AND	NOT	MM2VIS.bMsg3412
							AND	IN_SY.bCust_Dem_RSy;		(* release by customer *)

		END_IF;

		ton_mcb_dmnd_sy.PT := T#1s;
		ton_mcb_dmnd_sy();

		mcb.dmnd_sy	:=	ton_mcb_dmnd_sy.Q;

		(*----------------------------------------------------------------------------*)
		(* release trip mcb1 *)
		IF Para.bMCB_Enable THEN										(* mcb controlled by esy *)
			tof_mcb_rel_trip.IN :=	mcb.remote
								AND	bDem_Island
								AND	any_eng_run_bb;

		ELSE															(* mcb controlled by customer *)
			tof_mcb_rel_trip.IN :=	bDem_Island
								AND(IN_SY.tRel_Sync_Load.Do OR any_eng_run_bb);

		END_IF;

		tof_mcb_rel_trip.PT := T#1s;
		tof_mcb_rel_trip();

		mcb.rel_trip :=	tof_mcb_rel_trip.Q	AND	IN_SY.tPB2MM.bSys_Run;

		IF Para.bMCB_Enable THEN
			(*----------------------------------------------------------------------------*)
			(* monitoring release mcb *)
			mcb.mon_release :=	NOT mcb.alm_0sf
							AND	NOT	mcb.alm_1sf
							AND	NOT	mcb.alm_cf
							AND	NOT	mcb.alm_opf
							AND	NOT	mcb.alm_ol
							AND NOT ccb.alm_opf
							AND	NOT gcb_opf_delay;

			(*----------------------------------------------------------------------------*)
			(* release mcb *)
			mcb.release	:=	mcb.mon_release
					AND	NOT	OUT_SY.bOnly_Island
					AND		TRUE;										(* include additional release conditions *)

			(*----------------------------------------------------------------------------*)
			(* extend manual off command mcb *)
			tof_mcb_man_off(IN:= mcb.man_off, PT:= T#6s);

			(* extend demand synchronize mcb *)
			tof_mcb_dmnd_sy(IN:= mcb.dmnd_sy, PT:= T#100ms);

			(*----------------------------------------------------------------------------*)
			(* release close mcb *)
			ton_mcb_mrc.IN :=	NOT	MM2VIS.bMsg1216
							AND	NOT	gcb.dmnd_sy
							AND	NOT	any_gcb_psf_bb
							AND	NOT	mcb.alm_psf
							AND		IN_SY.tPB2MM.bSys_Run;

			ton_mcb_mrc.PT := T#6s;
			ton_mcb_mrc();

			mcb.mrc		  := ton_mcb_mrc.Q;

			(*----------------------------------------------------------------------------*)
//			VKE7			:=	all_gcb_off_bb
//						AND	NOT	mcb.on
//						AND		Para.bMCB_ReSw2Mns_Enable;

//			VKE8			:= (Para.bMCB_ReSw2Mns_Enable AND NOT mcb.on AND all_gcb_off_bb)
//							OR	bb_dead;

			(* manuell on mcb1 to dead busbar *)
			mcb_man_on2dead_bb :=	bSyOMSS_Man
							AND 	mcb.release
							AND 	mcb.remote
							AND 	mcb.rdy
							AND 	mcb.mrc
							AND 	mains.ok
							AND 	mcb.man_on
							AND	NOT	tof_mcb_man_off.Q
							AND	   (bb_dead OR (Para.bMCB_ReSw2Mns_Enable AND NOT mcb.on AND all_gcb_off_bb))
							AND NOT IN_SY.tDemGenExcOff.Di
							AND		IN_SY.tPB2MM.bSys_Run;

			mcb.man_on2dead_bb :=	mcb_man_on2dead_bb
							AND		rel_mcb_on2d_bb;

			(* automatic on mcb to dead busbar *)
			mcb_aut_on2dead_bb :=	bSyOMSS_Aut
							AND 	mcb.release
							AND 	mcb.remote
							AND 	mcb.rdy
							AND 	mcb.mrc
							AND 	mains.ok
							AND	   (bb_dead OR (Para.bMCB_ReSw2Mns_Enable AND NOT mcb.on AND all_gcb_off_bb))
							AND NOT IN_SY.tDemGenExcOff.Di
							AND		IN_SY.tPB2MM.bSys_Run;

			mcb.aut_on2dead_bb :=	mcb_aut_on2dead_bb
							AND		rel_mcb_on2d_bb;

			(*----------------------------------------------------------------------------*)
			(* release sy_puls mcb *)
			IF	Para.bMCB_ReSw2Mns_Enable THEN								(* reswitch  to mains *)
				mcb.rel_sy_puls :=	FALSE;
			ELSE															(* synchronization to mains *)
				mcb.rel_sy_puls :=	mcb.release
							AND		mcb.remote
							AND		tof_mcb_dmnd_sy.Q
							AND		IN_SY.tPB2MM.bSys_Run;
			END_IF;

			(*----------------------------------------------------------------------------*)
			(* command mcb off *)											(* OUT_SY.tMCB_COf.Do *)
			mcb.dmnd_off 	:=	mcb.remote
						AND(NOT mcb.release OR (tof_mcb_man_off.Q AND NOT bSyOMSS_Aut))
						AND		IN_SY.tPB2MM.bSys_Run;

			mcb.command_off :=	mcb.dmnd_off
						AND	NOT	mcb.off;

			(*----------------------------------------------------------------------------*)
			(* command mcb on *)
			mcb.dmnd_on		:=	mcb.remote
						AND		mcb.release
						AND    (mcb.aut_on2dead_bb OR mcb.man_on2dead_bb)
						AND		IN_SY.tPB2MM.bSys_Run;

			mcb.command_on	:=	mcb.dmnd_on
						AND	NOT	mcb.on
						AND	NOT	tof_mcb_man_off.Q;

			(*----------------------------------------------------------------------------*)
			(* release mcb1 (old hardware design) to delete after testing *)
		//	ton_einprns.IN :=
		//					NOT	mcb[3].release
		//				AND	NOT	mcb.signal_mon;
		//	ton_einprns.PT := T#5s;
		//	ton_einprns();
		//
		//	mcb[3].release	:=	mcb.monitoring_release
		//				AND(
		//				   (	mcb.mns_ok		OR	NOT	mcb.release_trip	)
		//				AND(	ton_einprns.Q	OR		mcb[3].release		)
		//				OR (
		//				   (NOT	mcb.remote		OR	NOT	IN_SY.tPB2MM.bSys_Run					)
		//				AND		all_gcb_off_bb									));
		//
		//	(* command mcb1 off (old hardware design) *)
		//	mcb[3].command_off :=
		//				   (	mcb[3].release		AND		bSyOMSS_Aut				)
		//				OR (	mcb[3].release		AND	NOT	tof_mcb_man_off.Q)
		//				OR (
		//				   (NOT	mcb.remote		OR	NOT	IN_SY.tPB2MM.bSys_Run					)
		//				AND		all_gcb_off_bb									);

			(*----------------------------------------------------------------------------*)

		END_IF;
	END_IF;

END_PROGRAM
```

#### mcb.var
```iecst
VAR
	tof_mcb_dmnd_sy : TOF;
	tof_mcb_man_off : TOF;
	tof_mcb_rel_trip : TOF;
	ton_mcb_dmnd_sy : TON;
	ton_mcb_mrc : TON;
END_VAR
```

### Program Logical/Synchronization/summary (IEC, version 2.60.0) - sy: summary

#### summaryCyclic.st
```iecst
(*******************************************************************************
SY: 	summary

This code is confidential and proprietary to the INNIO Company.
It may not be used in any form, or reproduced in any manner,
without the express written permission of the INNIO Company.
Copyright, INNIO Company, 2019

Customized modifications: -
------------------------

History:
-------
V1.10	12-01-2006	Lettenbichler, new
V1.11	16-03-2006	lettenbichler, customer gcb[0] added
V2.12	24.04.06/LH	adapted for esy new
		11.11.06/LH	revised after Para.bMSy test
V2.50.1 20.07.2009	lettenb.	any_gcb_opf_bb: OUT_SY.tGCB_OPF.Do added(temp.solution)
V2.60.0 13.08.2009	lettenb.	any_gcb_opf_bb: OUT_SY.tGCB_OPF.Do removed(temp.solution)

Instructions for use:
--------------------

Outstandings:
------------
*******************************************************************************)
PROGRAM _CYCLIC

	IF	Para.bSyActive THEN
		(*----------------------------------------------------------------------------*)
		other_gcb_on		:=	gcb.other_gcb_on	OR	ccb.on;			(* other gcb closed - busbar *)
		any_gcb_on_bb		:=	gcb.on				OR	other_gcb_on;	(* any   gcb closed - busbar *)

		other_gcb_off		:=	ccb.off	AND gcb.all_other_gcb_off;		(* other gcb opened - busbar *)
		all_gcb_off_bb		:=	gcb.off	AND	other_gcb_off;				(* all   gcb opened - busbar *)

		(*----------------------------------------------------------------------------*)
		any_eng_oper_and_gcb_on_bb	:= (ccb.eng_oper	AND	ccb.on)		(* any engine operating with closed gcb - busbar *)
									OR (gcb.eng_oper	AND	gcb.on);

		(*----------------------------------------------------------------------------*)
		OUT_SY.bOtherGenParallel	:=	gcb.other_gen_parallel 			(* any engine demanded and gcb on - busbar *)
									OR (ccb.eng_demanded	AND	ccb.on);

		(*----------------------------------------------------------------------------*)
		any_eng_run_bb		:=	gcb.eng_run	OR	ccb.eng_run;			(* any engine running - busbar *)
		no_eng_run_bb		:=	NOT	any_eng_run_bb;						(* no engine runing   - busbar *)

		(*----------------------------------------------------------------------------*)
		(* summary gcb alarms *)
		any_gcb_psf_bb		:=	gcb.alm_psf OR ccb.alm_psf;				(* any gcb position signal failure - busbar *)
		any_gcb_opf_bb		:=	gcb.alm_opf OR ccb.alm_opf;				(* any gcb opening failure         - busbar *)
		any_gcb_alarm_bb 	:=	gcb.alarm   OR ccb.alarm;				(* any gcb alarm                   - busbar *)

		(*----------------------------------------------------------------------------*)

	END_IF;

END_PROGRAM
```

### Program Logical/Synchronization/loadshedd (IEC, version 4.13.0) - loadshedding

#### loadsheddCyclic.st
```iecst
(***************************************************************************
loadshed			functions

This code is confidential and proprietary to the INNIO Company.
It may not be used in any form, or reproduced in any manner,
without the express written permission of the INNIO Company.
Copyright, INNIO Company, 2019

Customized modifications: -
------------------------

History:
-------
V0.1	10.07.1998 Pa			erstellt
 		24.11.1998 Pa			korrekturlesung
V170	08.03.2002 LH			Anforderung Netzstartgerät
 								Anforderung Entregung
 								Anforderung Lastabwurf
V180	21.03.2003 LH			Zuschaltung COSPHI-Regler geändert
V206	22.06.2004 LH			Freigabe Gemischregler über Parameter
V2071c	20.09.2005 LH			neu: Generator ohne Spannung
 								neu: Freigabe Spannungsanwahl LS-Generator
V2072	16.11.2005 LH			Grenzwert Generatorspannung auf Prozent Nennspannung bezogen
V190	14.04.2004 LH			Anforderung Lastabwurf angepasst
 		06.06.2006 LH			neu: Spannungsverstellung Generator
V2102	22.11.2006 LH			Lastabwurf durch Anforderung P-Reduktion im Inselbetrieb
 								GW Generatorspannung: 12,5% --> 30,0%
V212	16.10.2006 LH			Anpassungen für ESY-NEU
V220	19.02.2007 LH			E_LSHK nur noch für GSY aktiv
 								neu: Anforderung Heizwasserpumpe
 								neu: Quittierung Warnung
 		23.03.2007 LH			Aktivierung LSHK für CUN1 AvK-Generator (Plattner)
 		20.04.2007 LH			Eingabe Generator-Nennspannung --> settings
 		11.05.2007 LH			keine Entregung mehr beim Abstellvorgang (Kruckenhauser)
V2201	04.06.2007 LH			Anforderung Heizwasserpumpe --> Heizwasserpumpe EIN
V2225	23.04.2008 LH			Erweiterungen für Pakistan
V2.34.0	14.10.2008 lettenb.		generator deexcitation A_ENTR: M_GEN_PT added
V2.50.0	28.01.2009 lettenb.		M_MMD_OL added
								DO_DMND_LS: M_BTRB added for PAK
V2.60.0	07.08.2009 lettenb.		FA_A_QUITT from VISA added
V3.10.0	07.08.2009 lettenb.		A_COSPHI: PAK removed (country specific selection removed/steiger joh.)
								FG_KT: AN_RLT_M added (demand cooling tower/steiger/pfister)
V3.20.0	30.09.2010 maier(BuR)	M_GSEIN replaced with GCB_ON
								NS_EIN replaced with MCB_ON
		07.12.2010 lettenb.		DO_A_QUITT, DO_W_QUITT moved to task reset
		07.02.2011				FG_HGV, FG_HGV_ext release main gas valve added (moved from task biogas)
V3.30.0	20.10.2011 lettenb.		DMND_ICF added: demand charge cooler ventilation(intercooler fan)
V3.90.0	08.11.2011 lettenb.		new from pb8
V4.13.0 20.11.2023 Farre,		added IN_SY.bBypassMCB_LoadShed and request power mode interfaces from CU needed for Microgrid (2023-168)

Instructions for use:
--------------------

Outstandings:
------------
***************************************************************************)

PROGRAM _CYCLIC
	(*------------------------------------------------------------------------------------*)
	(* power maximum for load shedding *)
	xGR_MAXR_P_LS_Hi(In:= IN_SY.rP_Act_Norm_Filt, Gw:= Para.rP_LS_LimHi, Hy:= Para.rP_LS_HyHi);
	xTON_P_LS_Hi(IN:= xGR_MAXR_P_LS_Hi.Q AND IN_SY.tPB2MM.bParaSetupOk, PT:= Para.tiP_LS_LimHi);
	P_MAX := xTON_P_LS_Hi.Q;

	(*------------------------------------------------------------------------------------*)
	(* generator power low for load shedding warning *)
	xGR_MINR_P_LS_Lo(In:= IN_SY.rP_Act_Norm_Filt, Gw:= Para.rP_LS_LimLo, Hy:= Para.rP_LS_HyLo);
	xTON_P_LS_Lo(IN:= xGR_MINR_P_LS_Lo.Q AND IN_SY.tPB2MM.bParaSetupOk AND xOpMode.Island, PT:= Para.tiP_LS_LimLo);
	P_MIN_W := xTON_P_LS_Lo.Q;

	(*------------------------------------------------------------------------------------*)
	(* generator power low for load shedding trip *)
	xGR_MINR_P_LS_LoLo(In:= IN_SY.rP_Act_Norm_Filt, Gw:= Para.rP_LS_LimLoLo, Hy:= Para.rP_LS_HyLoLo);
	xTON_P_LS_LoLo(IN:= xGR_MINR_P_LS_LoLo.Q AND IN_SY.tPB2MM.bParaSetupOk AND xOpMode.Island, PT:= Para.tiP_LS_LimLoLo);
	P_MIN_A := xTON_P_LS_LoLo.Q;

	(*------------------------------------------------------------------------------------*)
	(* load shedding - engine speed limit low *)
	xGR_MINR_N_LS_Lo(In:= IN_SY.rN_EngAct, Gw:= Para.rN_LS_LimLo, Hy:= Para.rN_LS_HyLo);
	xTON_N_LS_Lo(IN:= xGR_MINR_N_LS_Lo.Q AND IN_SY.tPB2MM.bParaSetupOk, PT:= Para.tiN_LS_LimLo);
	DR_MIN := xTON_N_LS_Lo.Q;

	(*------------------------------------------------------------------------------------*)
	(*------------------------------------------------------------------------------*)
	OUT_SY.tN_EngStart.Do 	:= bN_EngStart;		(* M_DREHZ *)
	OUT_SY.tP_Lo.Do 		:= NOT bP_Lo;		// AN_LSA;

	(*------------------------------------------------------------------------------*)
	(* load shedding demand for island operation*)
	bLS4I_Dem :=	IN_SY.tGCB_On.Di
			AND ( NOT OUT_SY.bMCB_On OR IN_SY.bBypassMCB_LoadShed)
			AND(    P_MAX 				 OR     DR_MIN                   OR     IN_SY.bP_Red_Active)
			AND(NOT IN_SY.bReq_PowMod OR NOT OUT_SY.bOtherGenParallel OR NOT(Para.iCountry = iPakistan));

	(* load shedding demand for blackout start *)
	bLS4BL_Dem :=	BLOUT
			AND NOT OUT_SY.bOtherGenParallel
			AND    (IN_SY.tEng_Run.Do OR NOT (Para.iCountry = iPakistan));

	(* load shedding demand *)
	OUT_SY.tLS_Dem.Do := bLS4I_Dem OR bLS4BL_Dem;

	(*------------------------------------------------------------------------------*)

END_PROGRAM
```

#### loadshedd.var
```iecst
VAR
	xGR_MAXR_P_LS_Hi : GR_MAXR;
	xGR_MINR_P_LS_Lo : GR_MINR;
	xGR_MINR_P_LS_LoLo : GR_MINR;
	xGR_MINR_N_LS_Lo : GR_MINR;
	xTON_P_LS_Hi : TON;
	xTON_P_LS_Lo : TON;
	xTON_P_LS_LoLo : TON;
	xTON_N_LS_Lo : TON;
	bLS4I_Dem : BOOL;
	bLS4BL_Dem : BOOL;
END_VAR
```

### Program Logical/Synchronization/de_excit (IEC, version 4.13.0) - generator de-excitation
